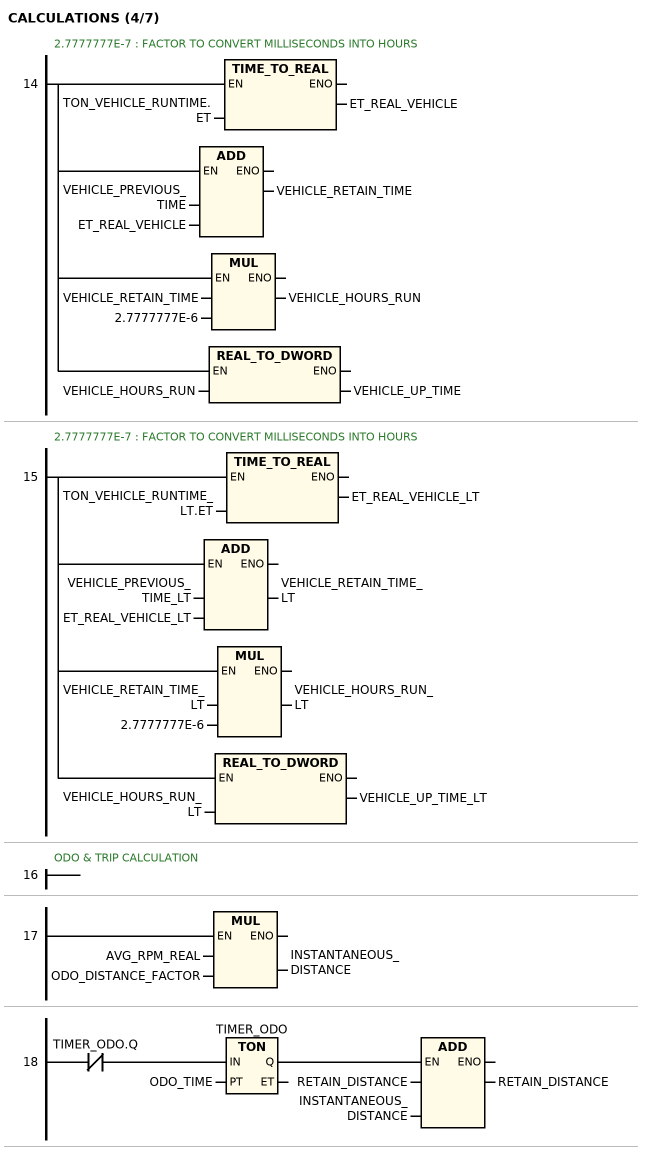
[picture p24: CALCULATIONS (LD)]
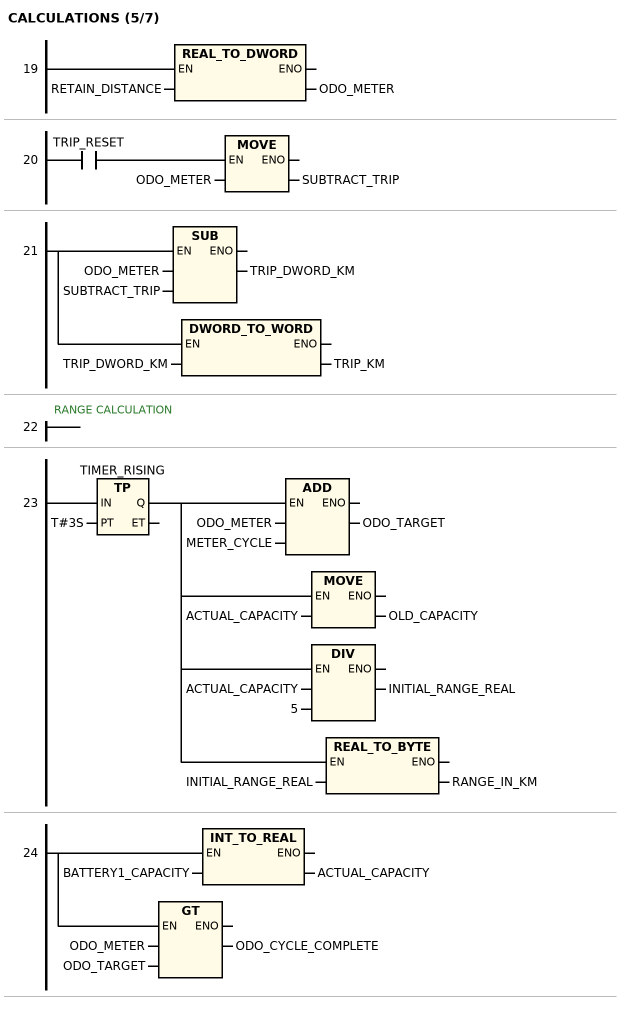
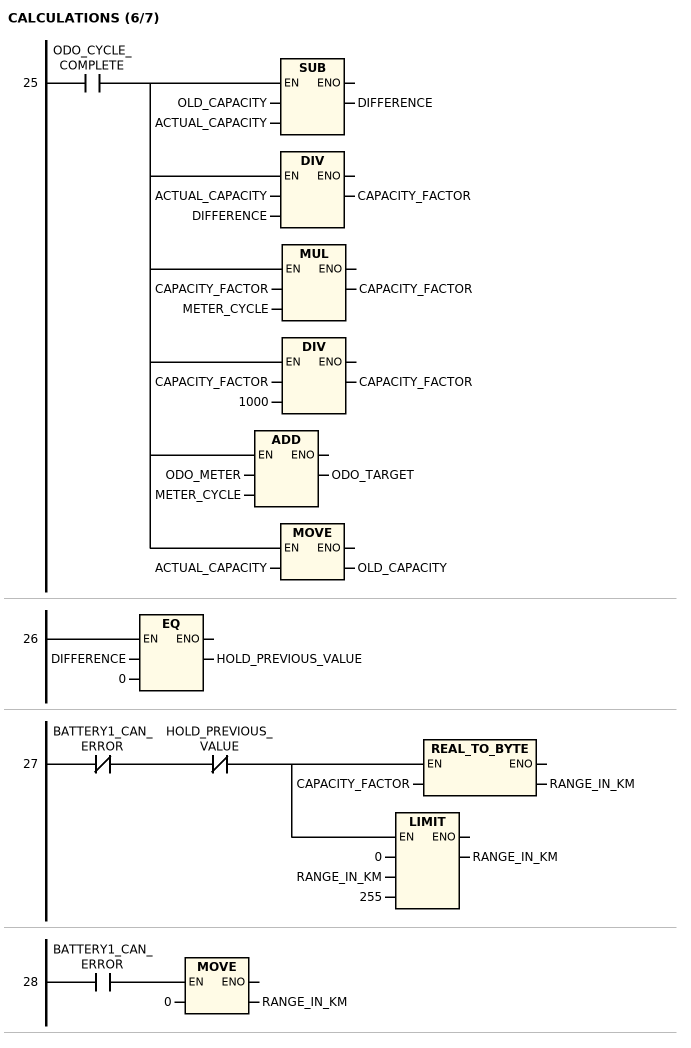
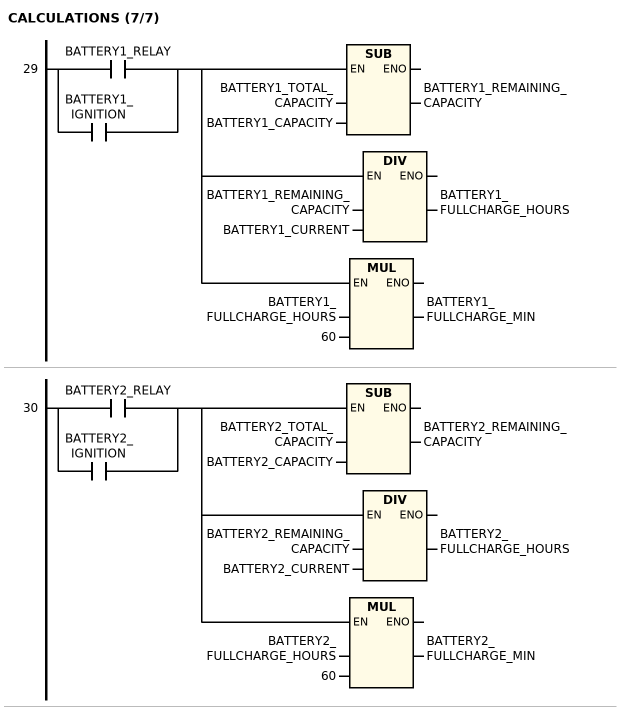
_LD_ (* Ladder Diagram *)
NETWORK 1 (* SPEED / GLX GEAR RATION = 72.02 / WHEEL DIA = 560 MM *)
	*
		EN --- ABS(MOTOR_RPM[1]) => ABS_RPM1
		EN --- ABS(MOTOR_RPM[2]) => ABS_RPM2
		EN --- ABS(MOTOR_RPM[6]) => ABS_RPM6
NETWORK 2
	*
		EN --- ADD(ABS_RPM1, ABS_RPM2) => RPM_SUM
		EN --- DIV(RPM_SUM, 2) => AVG_RPM
		EN --- ABS(AVG_RPM) => AVG_RPM
		EN --- INT_TO_REAL(AVG_RPM) => AVG_RPM_REAL
		EN --- MUL(AVG_RPM_REAL, SPEED_FACTOR) => SPEED_REAL
		EN --- REAL_TO_BYTE(SPEED_REAL) => SPEED
NETWORK 3 (* DRIVE AND HYDL UP TIME *)
	*
		EN --- GT(ABS_RPM1, 100) => MOTOR_1_RUNNING
		EN --- GT(ABS_RPM2, 100) => MOTOR_2_RUNNING
		EN --- OR(MOTOR_1_RUNNING, MOTOR_2_RUNNING) => COUNT_HOURS
		EN --- GT(ABS_RPM6, 100) => HYDRAULIC_HOURS
		EN --- OR(MCU_IGNITION, HYDRAULIC_SWITCH) => VEHICLE_UP_TIME_COUNT, VEHICLE_UP_TIME_COUNT_LT
NETWORK 4
	{ RISE:R_TRIG(CLK: *) | [COUNT_HOURS] - FALL:F_TRIG(CLK: *) }
		EN --- MOVE(RETAIN_TIME) => PREVIOUS_TIME
NETWORK 5
	{ RISE_2:R_TRIG(CLK: *) | [HYDRAULIC_HOURS] - FALL_2:F_TRIG(CLK: *) }
		EN --- MOVE(HYDL_RETAIN_TIME) => HYDL_PREVIOUS_TIME
NETWORK 6
	{ RISE_3:R_TRIG(CLK: *) | [VEHICLE_UP_TIME_COUNT] - FALL_3:F_TRIG(CLK: *) }
		EN --- MOVE(VEHICLE_RETAIN_TIME) => VEHICLE_PREVIOUS_TIME
NETWORK 7
	{ RISE_4:R_TRIG(CLK: *) | [VEHICLE_UP_TIME_COUNT_LT] - FALL_4:F_TRIG(CLK: *) }
		EN --- MOVE(VEHICLE_RETAIN_TIME_LT) => VEHICLE_PREVIOUS_TIME_LT
NETWORK 8
	[COUNT_HOURS] - TON_RUNTIME:TON(IN: *, PT: t#10d)
NETWORK 9
	[HYDRAULIC_HOURS] - TON_HYDL_RUNTIME:TON(IN: *, PT: t#10d)
NETWORK 10
	[VEHICLE_UP_TIME_COUNT] - TON_VEHICLE_RUNTIME:TON(IN: *, PT: t#10d)
NETWORK 11
	[VEHICLE_UP_TIME_COUNT_LT] - TON_VEHICLE_RUNTIME_LT:TON(IN: *, PT: t#10d)
NETWORK 12 (* 2.7777777E-6 : FACTOR TO CONVERT MILLISECONDS INTO (HOUR . MIN) (FACTOR IS 0.1) *)
	*
		EN --- TIME_TO_REAL(TON_RUNTIME.ET) => ET_REAL
		EN --- ADD(PREVIOUS_TIME, ET_REAL) => RETAIN_TIME
		EN --- MUL(RETAIN_TIME, 2.7777777E-6) => MINUTE_RUN
		EN --- REAL_TO_DWORD(MINUTE_RUN) => RUNTIME
NETWORK 13 (* 2.7777777E-7 : FACTOR TO CONVERT MILLISECONDS INTO HOURS *)
	*
		EN --- TIME_TO_REAL(TON_HYDL_RUNTIME.ET) => ET_REAL_HYDL
		EN --- ADD(HYDL_PREVIOUS_TIME, ET_REAL_HYDL) => HYDL_RETAIN_TIME
		EN --- MUL(HYDL_RETAIN_TIME, 2.7777777E-6) => HYDL_HOURS_RUN
		EN --- REAL_TO_DWORD(HYDL_HOURS_RUN) => HYDL_UP_TIME
NETWORK 14 (* 2.7777777E-7 : FACTOR TO CONVERT MILLISECONDS INTO HOURS *)
	*
		EN --- TIME_TO_REAL(TON_VEHICLE_RUNTIME.ET) => ET_REAL_VEHICLE
		EN --- ADD(VEHICLE_PREVIOUS_TIME, ET_REAL_VEHICLE) => VEHICLE_RETAIN_TIME
		EN --- MUL(VEHICLE_RETAIN_TIME, 2.7777777E-6) => VEHICLE_HOURS_RUN
		EN --- REAL_TO_DWORD(VEHICLE_HOURS_RUN) => VEHICLE_UP_TIME
NETWORK 15 (* 2.7777777E-7 : FACTOR TO CONVERT MILLISECONDS INTO HOURS *)
	*
		EN --- TIME_TO_REAL(TON_VEHICLE_RUNTIME_LT.ET) => ET_REAL_VEHICLE_LT
		EN --- ADD(VEHICLE_PREVIOUS_TIME_LT, ET_REAL_VEHICLE_LT) => VEHICLE_RETAIN_TIME_LT
		EN --- MUL(VEHICLE_RETAIN_TIME_LT, 2.7777777E-6) => VEHICLE_HOURS_RUN_LT
		EN --- REAL_TO_DWORD(VEHICLE_HOURS_RUN_LT) => VEHICLE_UP_TIME_LT
NETWORK 16 (* ODO & TRIP CALCULATION *)
	*
NETWORK 17
	*
		EN --- MUL(AVG_RPM_REAL, ODO_DISTANCE_FACTOR) => INSTANTANEOUS_DISTANCE
NETWORK 18
	[/TIMER_ODO.Q] - TIMER_ODO:TON(IN: *, PT: ODO_TIME)
		EN --- ADD(RETAIN_DISTANCE, INSTANTANEOUS_DISTANCE) => RETAIN_DISTANCE
NETWORK 19
	*
		EN --- REAL_TO_DWORD(RETAIN_DISTANCE) => ODO_METER
NETWORK 20
	[TRIP_RESET]
		EN --- MOVE(ODO_METER) => SUBTRACT_TRIP
NETWORK 21
	*
		EN --- SUB(ODO_METER, SUBTRACT_TRIP) => TRIP_DWORD_KM
		EN --- DWORD_TO_WORD(TRIP_DWORD_KM) => TRIP_KM
NETWORK 22 (* RANGE CALCULATION *)
	*
NETWORK 23
	TIMER_RISING:TP(IN: *, PT: T#3S)
		EN --- ADD(ODO_METER, METER_CYCLE) => ODO_TARGET
		EN --- MOVE(ACTUAL_CAPACITY) => OLD_CAPACITY
		EN --- DIV(ACTUAL_CAPACITY, 5) => INITIAL_RANGE_REAL
		EN --- REAL_TO_BYTE(INITIAL_RANGE_REAL) => RANGE_IN_KM
NETWORK 24
	*
		EN --- INT_TO_REAL(BATTERY1_CAPACITY) => ACTUAL_CAPACITY
		EN --- GT(ODO_METER, ODO_TARGET) => ODO_CYCLE_COMPLETE
NETWORK 25
	[ODO_CYCLE_COMPLETE]
		EN --- SUB(OLD_CAPACITY, ACTUAL_CAPACITY) => DIFFERENCE
		EN --- DIV(ACTUAL_CAPACITY, DIFFERENCE) => CAPACITY_FACTOR
		EN --- MUL(CAPACITY_FACTOR, METER_CYCLE) => CAPACITY_FACTOR
		EN --- DIV(CAPACITY_FACTOR, 1000) => CAPACITY_FACTOR
		EN --- ADD(ODO_METER, METER_CYCLE) => ODO_TARGET
		EN --- MOVE(ACTUAL_CAPACITY) => OLD_CAPACITY
NETWORK 26
	*
		EN --- EQ(DIFFERENCE, 0) => HOLD_PREVIOUS_VALUE
NETWORK 27
	[/BATTERY1_CAN_ERROR] - [/HOLD_PREVIOUS_VALUE]
		EN --- REAL_TO_BYTE(CAPACITY_FACTOR) => RANGE_IN_KM
		EN --- LIMIT(0, RANGE_IN_KM, 255) => RANGE_IN_KM
NETWORK 28
	[BATTERY1_CAN_ERROR]
		EN --- MOVE(0) => RANGE_IN_KM
NETWORK 29
	{ [BATTERY1_RELAY] | [BATTERY1_IGNITION] }
		EN --- SUB(BATTERY1_TOTAL_CAPACITY, BATTERY1_CAPACITY) => BATTERY1_REMAINING_CAPACITY
		EN --- DIV(BATTERY1_REMAINING_CAPACITY, BATTERY1_CURRENT) => BATTERY1_FULLCHARGE_HOURS
		EN --- MUL(BATTERY1_FULLCHARGE_HOURS, 60) => BATTERY1_FULLCHARGE_MIN
NETWORK 30
	{ [BATTERY2_RELAY] | [BATTERY2_IGNITION] }
		EN --- SUB(BATTERY2_TOTAL_CAPACITY, BATTERY2_CAPACITY) => BATTERY2_REMAINING_CAPACITY
		EN --- DIV(BATTERY2_REMAINING_CAPACITY, BATTERY2_CURRENT) => BATTERY2_FULLCHARGE_HOURS
		EN --- MUL(BATTERY2_FULLCHARGE_HOURS, 60) => BATTERY2_FULLCHARGE_MIN
_END_LD_
(* the same logic as Structured Text *)
(* Network 1 *)
ABS_RPM1 := ABS(MOTOR_RPM[1]);
ABS_RPM2 := ABS(MOTOR_RPM[2]);
ABS_RPM6 := ABS(MOTOR_RPM[6]);
(* Network 2 *)
RPM_SUM := ABS_RPM1 + ABS_RPM2;
AVG_RPM := RPM_SUM / 2;
AVG_RPM := ABS(AVG_RPM);
AVG_RPM_REAL := INT_TO_REAL(AVG_RPM);
SPEED_REAL := AVG_RPM_REAL * SPEED_FACTOR;
SPEED := REAL_TO_BYTE(SPEED_REAL);
(* Network 3: see the listing above *)
(* Network 4 *)
RISE(CLK := TRUE);
FALL(CLK := COUNT_HOURS);
IF RISE.Q OR FALL.Q THEN
	PREVIOUS_TIME := RETAIN_TIME;
END_IF;
(* Network 5 *)
RISE_2(CLK := TRUE);
FALL_2(CLK := HYDRAULIC_HOURS);
IF RISE_2.Q OR FALL_2.Q THEN
	HYDL_PREVIOUS_TIME := HYDL_RETAIN_TIME;
END_IF;
(* Network 6 *)
RISE_3(CLK := TRUE);
FALL_3(CLK := VEHICLE_UP_TIME_COUNT);
IF RISE_3.Q OR FALL_3.Q THEN
	VEHICLE_PREVIOUS_TIME := VEHICLE_RETAIN_TIME;
END_IF;
(* Network 7 *)
RISE_4(CLK := TRUE);
FALL_4(CLK := VEHICLE_UP_TIME_COUNT_LT);
IF RISE_4.Q OR FALL_4.Q THEN
	VEHICLE_PREVIOUS_TIME_LT := VEHICLE_RETAIN_TIME_LT;
END_IF;
(* Network 8 *)
TON_RUNTIME(IN := COUNT_HOURS, PT := t#10d);
(* Network 9 *)
TON_HYDL_RUNTIME(IN := HYDRAULIC_HOURS, PT := t#10d);
(* Network 10 *)
TON_VEHICLE_RUNTIME(IN := VEHICLE_UP_TIME_COUNT, PT := t#10d);
(* Network 11 *)
TON_VEHICLE_RUNTIME_LT(IN := VEHICLE_UP_TIME_COUNT_LT, PT := t#10d);
(* Network 12 *)
ET_REAL := TIME_TO_REAL(TON_RUNTIME.ET);
RETAIN_TIME := PREVIOUS_TIME + ET_REAL;
MINUTE_RUN := RETAIN_TIME * (2.7777777E-6);
RUNTIME := REAL_TO_DWORD(MINUTE_RUN);
(* Network 13 *)
ET_REAL_HYDL := TIME_TO_REAL(TON_HYDL_RUNTIME.ET);
HYDL_RETAIN_TIME := HYDL_PREVIOUS_TIME + ET_REAL_HYDL;
HYDL_HOURS_RUN := HYDL_RETAIN_TIME * (2.7777777E-6);
HYDL_UP_TIME := REAL_TO_DWORD(HYDL_HOURS_RUN);
(* Network 14 *)
ET_REAL_VEHICLE := TIME_TO_REAL(TON_VEHICLE_RUNTIME.ET);
VEHICLE_RETAIN_TIME := VEHICLE_PREVIOUS_TIME + ET_REAL_VEHICLE;
VEHICLE_HOURS_RUN := VEHICLE_RETAIN_TIME * (2.7777777E-6);
VEHICLE_UP_TIME := REAL_TO_DWORD(VEHICLE_HOURS_RUN);
(* Network 15 *)
ET_REAL_VEHICLE_LT := TIME_TO_REAL(TON_VEHICLE_RUNTIME_LT.ET);
VEHICLE_RETAIN_TIME_LT := VEHICLE_PREVIOUS_TIME_LT + ET_REAL_VEHICLE_LT;
VEHICLE_HOURS_RUN_LT := VEHICLE_RETAIN_TIME_LT * (2.7777777E-6);
VEHICLE_UP_TIME_LT := REAL_TO_DWORD(VEHICLE_HOURS_RUN_LT);
(* Network 16: see the listing above *)
(* Network 17 *)
INSTANTANEOUS_DISTANCE := AVG_RPM_REAL * ODO_DISTANCE_FACTOR;
(* Network 18 *)
TIMER_ODO(IN := NOT TIMER_ODO.Q, PT := ODO_TIME);
IF TIMER_ODO.Q THEN
	RETAIN_DISTANCE := RETAIN_DISTANCE + INSTANTANEOUS_DISTANCE;
END_IF;
(* Network 19 *)
ODO_METER := REAL_TO_DWORD(RETAIN_DISTANCE);
(* Network 20 *)
IF TRIP_RESET THEN
	SUBTRACT_TRIP := ODO_METER;
END_IF;
(* Network 21 *)
TRIP_DWORD_KM := ODO_METER - SUBTRACT_TRIP;
TRIP_KM := DWORD_TO_WORD(TRIP_DWORD_KM);
(* Network 22: see the listing above *)
(* Network 23 *)
TIMER_RISING(IN := TRUE, PT := T#3S);
IF TIMER_RISING.Q THEN
	ODO_TARGET := ODO_METER + METER_CYCLE;
	OLD_CAPACITY := ACTUAL_CAPACITY;
	INITIAL_RANGE_REAL := ACTUAL_CAPACITY / 5;
	RANGE_IN_KM := REAL_TO_BYTE(INITIAL_RANGE_REAL);
END_IF;
(* Network 24 *)
ACTUAL_CAPACITY := INT_TO_REAL(BATTERY1_CAPACITY);
ODO_CYCLE_COMPLETE := ODO_METER > ODO_TARGET;
(* Network 25 *)
IF ODO_CYCLE_COMPLETE THEN
	DIFFERENCE := OLD_CAPACITY - ACTUAL_CAPACITY;
	CAPACITY_FACTOR := ACTUAL_CAPACITY / DIFFERENCE;
	CAPACITY_FACTOR := CAPACITY_FACTOR * METER_CYCLE;
	CAPACITY_FACTOR := CAPACITY_FACTOR / 1000;
	ODO_TARGET := ODO_METER + METER_CYCLE;
	OLD_CAPACITY := ACTUAL_CAPACITY;
END_IF;
(* Network 26 *)
HOLD_PREVIOUS_VALUE := DIFFERENCE = 0;
(* Network 27 *)
IF NOT BATTERY1_CAN_ERROR AND NOT HOLD_PREVIOUS_VALUE THEN
	RANGE_IN_KM := REAL_TO_BYTE(CAPACITY_FACTOR);
	RANGE_IN_KM := LIMIT(0, RANGE_IN_KM, 255);
END_IF;
(* Network 28 *)
IF BATTERY1_CAN_ERROR THEN
	RANGE_IN_KM := 0;
END_IF;
(* Network 29 *)
IF BATTERY1_RELAY OR BATTERY1_IGNITION THEN
	BATTERY1_REMAINING_CAPACITY := BATTERY1_TOTAL_CAPACITY - BATTERY1_CAPACITY;
	BATTERY1_FULLCHARGE_HOURS := BATTERY1_REMAINING_CAPACITY / BATTERY1_CURRENT;
	BATTERY1_FULLCHARGE_MIN := BATTERY1_FULLCHARGE_HOURS * 60;
END_IF;
(* Network 30 *)
IF BATTERY2_RELAY OR BATTERY2_IGNITION THEN
	BATTERY2_REMAINING_CAPACITY := BATTERY2_TOTAL_CAPACITY - BATTERY2_CAPACITY;
	BATTERY2_FULLCHARGE_HOURS := BATTERY2_REMAINING_CAPACITY / BATTERY2_CURRENT;
	BATTERY2_FULLCHARGE_MIN := BATTERY2_FULLCHARGE_HOURS * 60;
END_IF;
END_PROGRAM

(* POU FB_LIBRARY/ALTERNATE, LD *)
FUNCTION_BLOCK ALTERNATE
VAR_INPUT
	IN: BOOL;
END_VAR
VAR_OUTPUT
	OUT: BOOL;
END_VAR
VAR
	S1: BOOL;
	S2: BOOL;
END_VAR
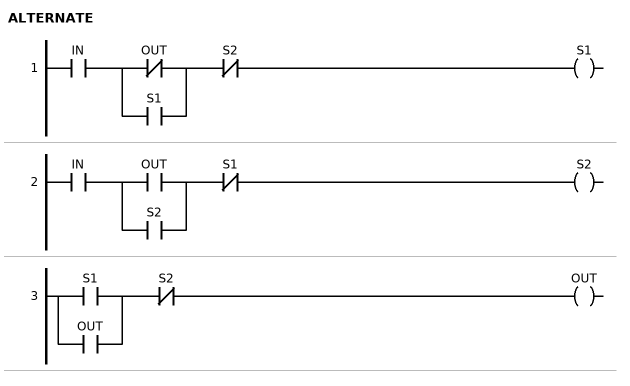
_LD_ (* Ladder Diagram *)
NETWORK 1
	[IN] - { [/OUT] | [S1] } - [/S2] --- (S1)
NETWORK 2
	[IN] - { [OUT] | [S2] } - [/S1] --- (S2)
NETWORK 3
	{ [S1] | [OUT] } - [/S2] --- (OUT)
_END_LD_
(* the same logic as Structured Text *)
(* Network 1 *)
S1 := IN AND (NOT OUT OR S1) AND NOT S2;
(* Network 2 *)
S2 := IN AND (OUT OR S2) AND NOT S1;
(* Network 3 *)
OUT := (S1 OR OUT) AND NOT S2;
END_FUNCTION_BLOCK

(* POU PROGRAM_FBs/ARM_LOGIC, LD *)
FUNCTION_BLOCK ARM_LOGIC
VAR_INPUT
	ARM_INPUT: BOOL;
	DISARM: BOOL;
	POST_IN: BOOL;
END_VAR
VAR_OUTPUT
	ARM: BOOL;
	ARMLED: BOOL;
END_VAR
VAR
	DELAY: TON;
	S1: BOOL;
	S2: BOOL;
	BLINKY: BLINK;
END_VAR
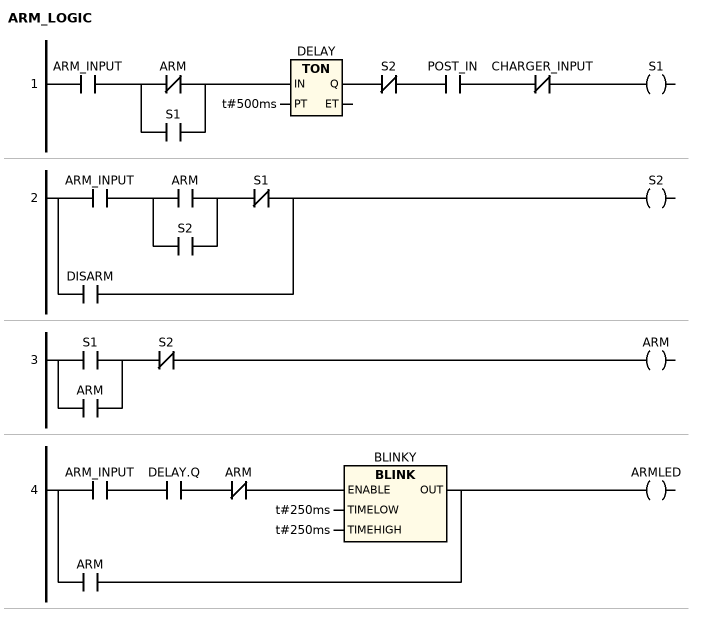
_LD_ (* Ladder Diagram *)
NETWORK 1
	[ARM_INPUT] - { [/ARM] | [S1] } - DELAY:TON(IN: *, PT: t#500ms) - [/S2] - [POST_IN] - [/CHARGER_INPUT] --- (S1)
NETWORK 2
	{ [ARM_INPUT] - { [ARM] | [S2] } - [/S1] | [DISARM] } --- (S2)
NETWORK 3
	{ [S1] | [ARM] } - [/S2] --- (ARM)
NETWORK 4
	{ [ARM_INPUT] - [DELAY.Q] - [/ARM] - BLINKY:BLINK(ENABLE: *, TIMELOW: t#250ms, TIMEHIGH: t#250ms) | [ARM] } --- (ARMLED)
_END_LD_
(* the same logic as Structured Text *)
(* Network 1 *)
DELAY(IN := ARM_INPUT AND (NOT ARM OR S1), PT := t#500ms);
S1 := DELAY.Q AND NOT S2 AND POST_IN AND NOT CHARGER_INPUT;
(* Network 2 *)
S2 := ARM_INPUT AND (ARM OR S2) AND NOT S1 OR DISARM;
(* Network 3 *)
ARM := (S1 OR ARM) AND NOT S2;
(* Network 4 *)
BLINKY(ENABLE := ARM_INPUT AND DELAY.Q AND NOT ARM, TIMELOW := t#250ms, TIMEHIGH := t#250ms);
ARMLED := BLINKY.OUT OR ARM;
END_FUNCTION_BLOCK

(* POU FUNCTIONS/BYTE_WORD_FUNCTION, ST *)
FUNCTION BYTE_WORD_FUNCTION : WORD
(*
Created by: Bhagyesh Unadkat
Date: 29-03-24
Version: 1
Updated by:
Update date:
Description: This block merges Two bytes of data into WORD data.
*)
VAR_INPUT
	BYTE_H: BYTE;
	BYTE_L: BYTE;
END_VAR
VAR
	MSB: WORD;
END_VAR
MSB:= BYTE_H * 256;
BYTE_WORD_FUNCTION:= MSB + BYTE_L;
END_FUNCTION

(* POU MCU/CHARA_MCU_RX, LD *)
FUNCTION_BLOCK CHARA_MCU_RX
(*
Created by: Bhagyesh Unadkat
Date: 11-09-24
Version: 5
Updated by: Karthik
Update date: 08-03-25
Description: This block receives CAN data from CHARA MCU.

		***Updates***
V2
	DC current and POWER added.
V3   
	Added OBD Code and adjusted the fault array accordingly.
	CAN error added to OBD code MSB bit as it is 12-bit value.
V4 
	Taken Motor Ignition as VAR_INPUT to reset RPM AND POWER TO 0
V5
	Converted CURRENT raw values from word to int, and then dividing by 1000.
V6
	Unmerged CAN error and OBD code.
V7
	Making OBD code zero when theres is a CAN error. 

FAULT ARRAY [DATATYPE: BYTE]
[1] MSG-2 BYTE2 and MSG-5 BYTE3		
		BYTE [BIT 0..7]: MSG2BYTE2 (BIT_0 TO BIT_2)------- AND-------- MSG5BYTE3 (BIT_0 TO BIT_4)
[2] MSG 2 :BYTE 7
[3] MSG 5: BYTE 2
[4] MSG 5: BYTE 4
*)
VAR_INPUT
	IGNITION: BOOL;
	MOTOR_IGNITION: BOOL;
	CAN_CHANNEL: BYTE;
	ID_1: DWORD;
	ID_2: DWORD;
	ID_4: DWORD;
	ID_5: DWORD;
	ID_6: DWORD;
END_VAR
VAR_OUTPUT
	RPM: INT;
	POWER: INT;
	PHASE_CURRENT: WORD;
	M_TEMP: BYTE;
	C_TEMP: BYTE;
	OBD_CODE: WORD;
	FAULT_ARRAY: ARRAY [1..4] OF BYTE;
	CAN_ERROR: BOOL;
END_VAR
VAR
	RX_1: RX_CAN;
	RX_2: RX_CAN;
	RX_4: RX_CAN;
	RX_5: RX_CAN;
	RX_6: RX_CAN;
	TIMER_ERROR: TON;

	RPM_WORD: WORD;
	PHASE_WORD: WORD;
	REVERSE_DIRECTION: BOOL;
	DIR_FACTOR: INT;
	DELAY: TON;
	RPM_INT: INT;
	CURRENT_WORD: WORD;
	CURRENT_INT: INT;
	VOLTAGE_INT: INT;
	RPM_SIGNED: INT;
	POWER_INT: INT;
END_VAR
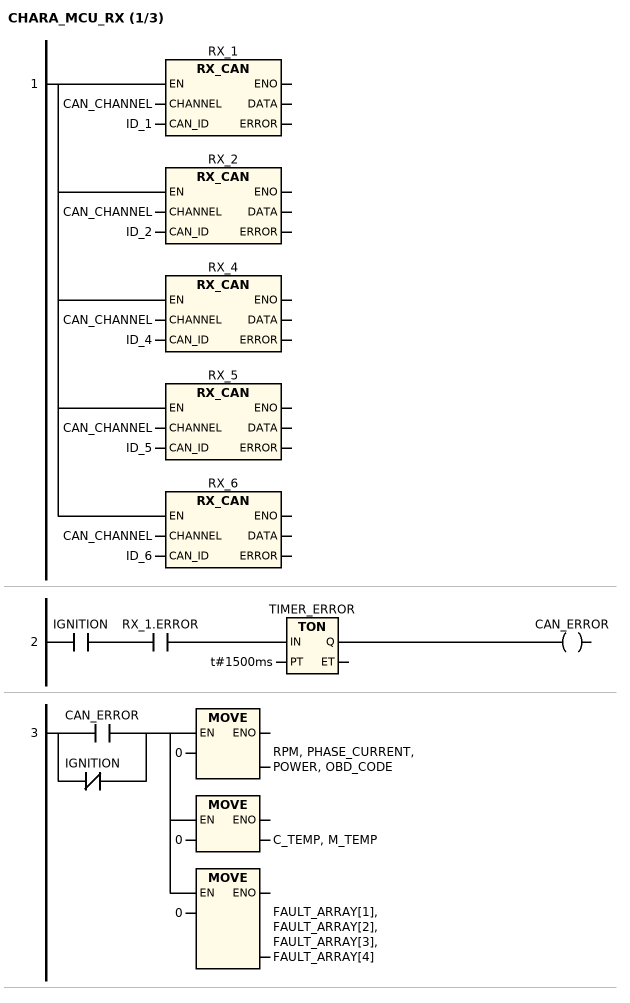
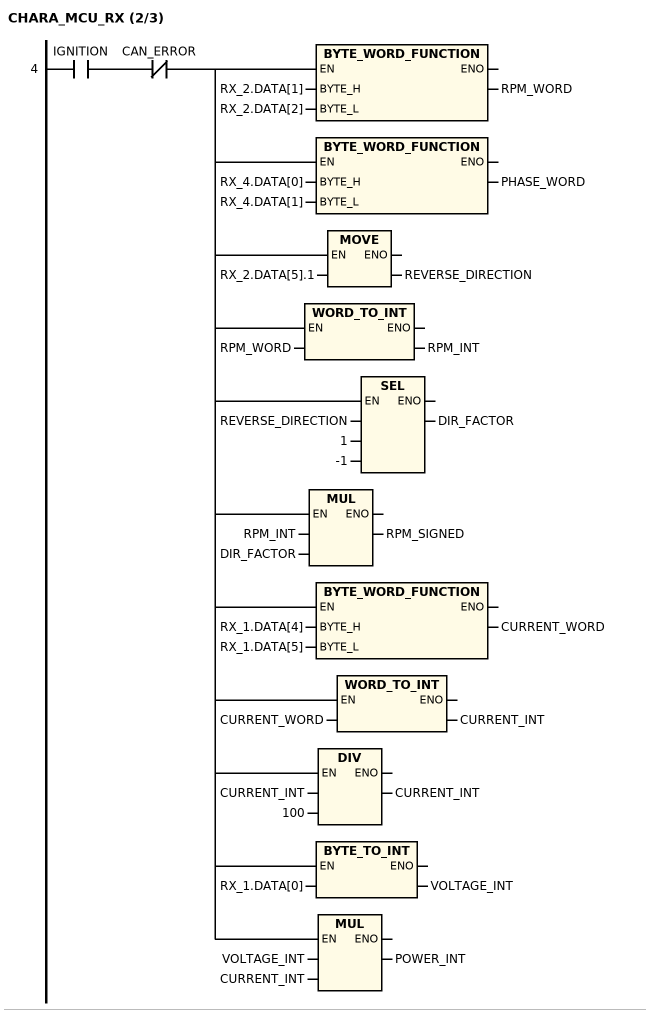
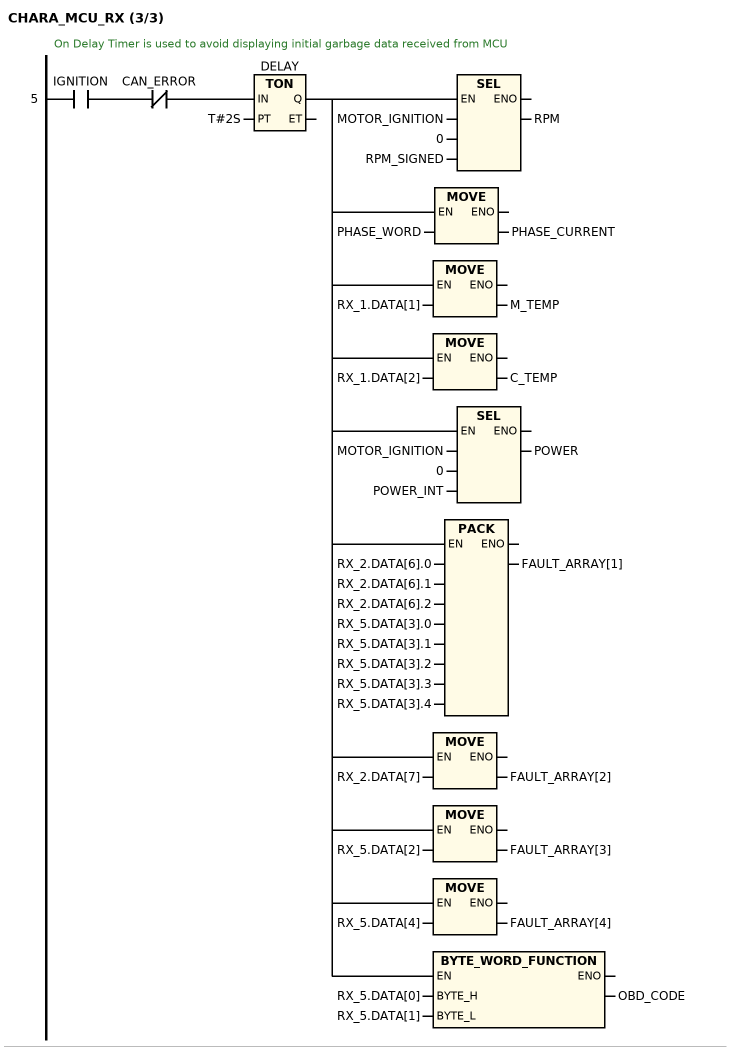
_LD_ (* Ladder Diagram *)
NETWORK 1
	*
		EN --- RX_1:RX_CAN(CHANNEL: CAN_CHANNEL, CAN_ID: ID_1)
		EN --- RX_2:RX_CAN(CHANNEL: CAN_CHANNEL, CAN_ID: ID_2)
		EN --- RX_4:RX_CAN(CHANNEL: CAN_CHANNEL, CAN_ID: ID_4)
		EN --- RX_5:RX_CAN(CHANNEL: CAN_CHANNEL, CAN_ID: ID_5)
		EN --- RX_6:RX_CAN(CHANNEL: CAN_CHANNEL, CAN_ID: ID_6)
NETWORK 2
	[IGNITION] - [RX_1.ERROR] - TIMER_ERROR:TON(IN: *, PT: t#1500ms) --- (CAN_ERROR)
NETWORK 3
	{ [CAN_ERROR] | [/IGNITION] }
		EN --- MOVE(0) => RPM, PHASE_CURRENT, POWER, OBD_CODE
		EN --- MOVE(0) => C_TEMP, M_TEMP
		EN --- MOVE(0) => FAULT_ARRAY[1], FAULT_ARRAY[2], FAULT_ARRAY[3], FAULT_ARRAY[4]
NETWORK 4
	[IGNITION] - [/CAN_ERROR]
		EN --- BYTE_WORD_FUNCTION(BYTE_H: RX_2.DATA[1], BYTE_L: RX_2.DATA[2]) => RPM_WORD
		EN --- BYTE_WORD_FUNCTION(BYTE_H: RX_4.DATA[0], BYTE_L: RX_4.DATA[1]) => PHASE_WORD
		EN --- MOVE(RX_2.DATA[5].1) => REVERSE_DIRECTION
		EN --- WORD_TO_INT(RPM_WORD) => RPM_INT
		EN --- SEL(REVERSE_DIRECTION, 1, -1) => DIR_FACTOR
		EN --- MUL(RPM_INT, DIR_FACTOR) => RPM_SIGNED
		EN --- BYTE_WORD_FUNCTION(BYTE_H: RX_1.DATA[4], BYTE_L: RX_1.DATA[5]) => CURRENT_WORD
		EN --- WORD_TO_INT(CURRENT_WORD) => CURRENT_INT
		EN --- DIV(CURRENT_INT, 100) => CURRENT_INT
		EN --- BYTE_TO_INT(RX_1.DATA[0]) => VOLTAGE_INT
		EN --- MUL(VOLTAGE_INT, CURRENT_INT) => POWER_INT
NETWORK 5 (* On Delay Timer is used to avoid displaying initial garbage data received from MCU *)
	[IGNITION] - [/CAN_ERROR] - DELAY:TON(IN: *, PT: T#2S)
		EN --- SEL(MOTOR_IGNITION, 0, RPM_SIGNED) => RPM
		EN --- MOVE(PHASE_WORD) => PHASE_CURRENT
		EN --- MOVE(RX_1.DATA[1]) => M_TEMP
		EN --- MOVE(RX_1.DATA[2]) => C_TEMP
		EN --- SEL(MOTOR_IGNITION, 0, POWER_INT) => POWER
		EN --- PACK(RX_2.DATA[6].0, RX_2.DATA[6].1, RX_2.DATA[6].2, RX_5.DATA[3].0, RX_5.DATA[3].1, RX_5.DATA[3].2, RX_5.DATA[3].3, RX_5.DATA[3].4) => FAULT_ARRAY[1]
		EN --- MOVE(RX_2.DATA[7]) => FAULT_ARRAY[2]
		EN --- MOVE(RX_5.DATA[2]) => FAULT_ARRAY[3]
		EN --- MOVE(RX_5.DATA[4]) => FAULT_ARRAY[4]
		EN --- BYTE_WORD_FUNCTION(BYTE_H: RX_5.DATA[0], BYTE_L: RX_5.DATA[1]) => OBD_CODE
_END_LD_
(* the same logic as Structured Text *)
(* Network 1 *)
RX_1(CHANNEL := CAN_CHANNEL, CAN_ID := ID_1);
RX_2(CHANNEL := CAN_CHANNEL, CAN_ID := ID_2);
RX_4(CHANNEL := CAN_CHANNEL, CAN_ID := ID_4);
RX_5(CHANNEL := CAN_CHANNEL, CAN_ID := ID_5);
RX_6(CHANNEL := CAN_CHANNEL, CAN_ID := ID_6);
(* Network 2 *)
TIMER_ERROR(IN := IGNITION AND RX_1.ERROR, PT := t#1500ms);
CAN_ERROR := TIMER_ERROR.Q;
(* Network 3: see the listing above *)
(* Network 4 *)
IF IGNITION AND NOT CAN_ERROR THEN
	RPM_WORD := BYTE_WORD_FUNCTION(BYTE_H := RX_2.DATA[1], BYTE_L := RX_2.DATA[2]);
	PHASE_WORD := BYTE_WORD_FUNCTION(BYTE_H := RX_4.DATA[0], BYTE_L := RX_4.DATA[1]);
	REVERSE_DIRECTION := RX_2.DATA[5].1;
	RPM_INT := WORD_TO_INT(RPM_WORD);
	DIR_FACTOR := SEL(REVERSE_DIRECTION, 1, -1);
	RPM_SIGNED := RPM_INT * DIR_FACTOR;
	CURRENT_WORD := BYTE_WORD_FUNCTION(BYTE_H := RX_1.DATA[4], BYTE_L := RX_1.DATA[5]);
	CURRENT_INT := WORD_TO_INT(CURRENT_WORD);
	CURRENT_INT := CURRENT_INT / 100;
	VOLTAGE_INT := BYTE_TO_INT(RX_1.DATA[0]);
	POWER_INT := VOLTAGE_INT * CURRENT_INT;
END_IF;
(* Network 5 *)
DELAY(IN := IGNITION AND NOT CAN_ERROR, PT := T#2S);
IF DELAY.Q THEN
	RPM := SEL(MOTOR_IGNITION, 0, RPM_SIGNED);
	PHASE_CURRENT := PHASE_WORD;
	M_TEMP := RX_1.DATA[1];
	C_TEMP := RX_1.DATA[2];
	POWER := SEL(MOTOR_IGNITION, 0, POWER_INT);
	FAULT_ARRAY[1] := PACK(RX_2.DATA[6].0, RX_2.DATA[6].1, RX_2.DATA[6].2, RX_5.DATA[3].0, RX_5.DATA[3].1, RX_5.DATA[3].2, RX_5.DATA[3].3, RX_5.DATA[3].4);
	FAULT_ARRAY[2] := RX_2.DATA[7];
	FAULT_ARRAY[3] := RX_5.DATA[2];
	FAULT_ARRAY[4] := RX_5.DATA[4];
	OBD_CODE := BYTE_WORD_FUNCTION(BYTE_H := RX_5.DATA[0], BYTE_L := RX_5.DATA[1]);
END_IF;
END_FUNCTION_BLOCK

(* POU MCU/CHARA_MCU_TX, LD *)
FUNCTION_BLOCK CHARA_MCU_TX
(*
Created by: Bhagyesh Unadkat
Date: Sep 11, 2024
Version: 4
Updated by: Bhagyesh
Update date: Dec 13, 2024
Description: This block transmits CAN data to the CHARA MCU to control the motor.

NOTE:  BIG ENDIAN FORMAT

Byte0 & Byte1: Signed RPM Big Endian format (-6000 to 6000)
Byte2: Ignition State =  0 & 1 (OFF and ON respectively)
Byte3: Phase Current Limit (%) = 0 - 100
Byte4: Regen (%) = 0 - 100 (Not configured yet)
Byte5: Acceleration time (s) = 1 unit is 100ms
Byte6: Deceleration time (s) =  1 unit is 100ms

CAN ID X value for the different Node ID:
41 - 9		42 - A 		43-B
	
	***UPDATES***
V2:
1. RPM transmit delay has been added after Ignition turns on..
2. CAN_TX block has been changerd to CAN_TX_ENH.
3. Temporary Phase current limit has been added to var input
V3
1. Added Ignition state bit as VAR_OUTPUT.
V4
1. UPDATED AVG RPM TO 75 TO HOLD ON THE MCU.
2. RPM DELAY TIME REDUCED TO 250MS
*)
VAR_INPUT
	CAN_CHANNEL: BYTE;
	ID_22X: DWORD;
	TARGET_RPM: INT;
	REFERNCE_RPM: INT;
	RAMP: INT;
	MCU_RAMP: BYTE;
	HILL_HOLD_IN: BOOL;
	PHASE_CURRENT_LIMIT: BYTE;
END_VAR
VAR
	IGNITION_ON: BOOL;
	IGNITION_STATE: BYTE;
	HOLD_ON: BOOL;
	ABS_RPM: INT;
	RPM_RAMP: RAMP_INT;
	WB_TARGET_RPM: WORD_BYTE_CONVERSION;
	PACK_TX: PACK_BYTES;
	TX: CAN_TX_ENH;
	RPM_DELAY: TON;
	TIMER: TON;
END_VAR
VAR_OUTPUT
	TARGET_RPM_OUT: INT;
	IGNITION_OUT: BOOL;
END_VAR
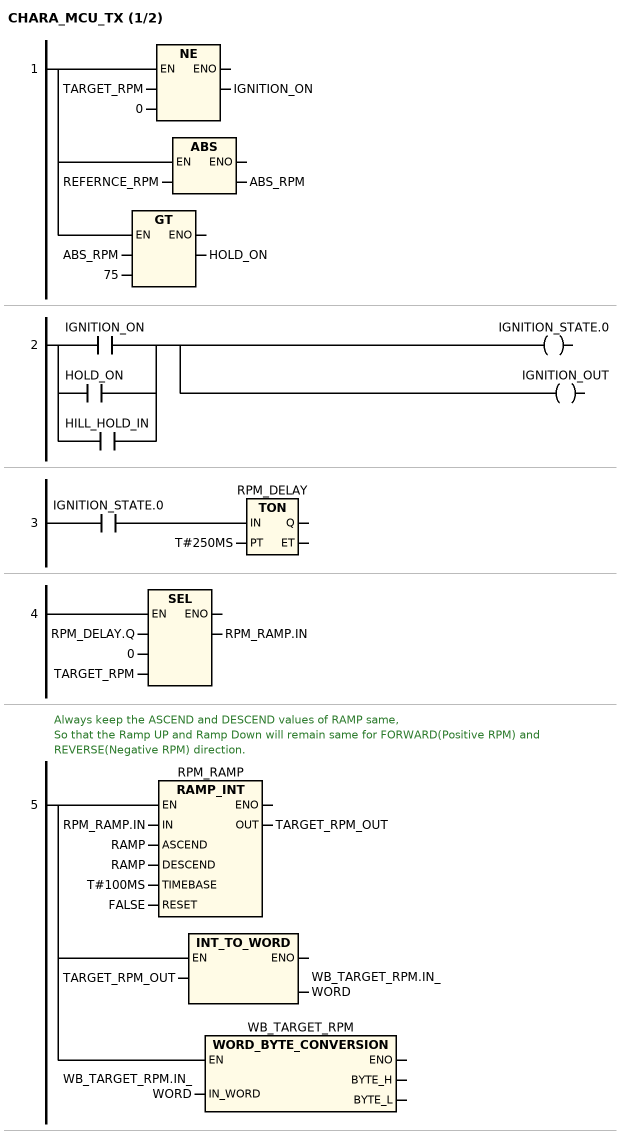
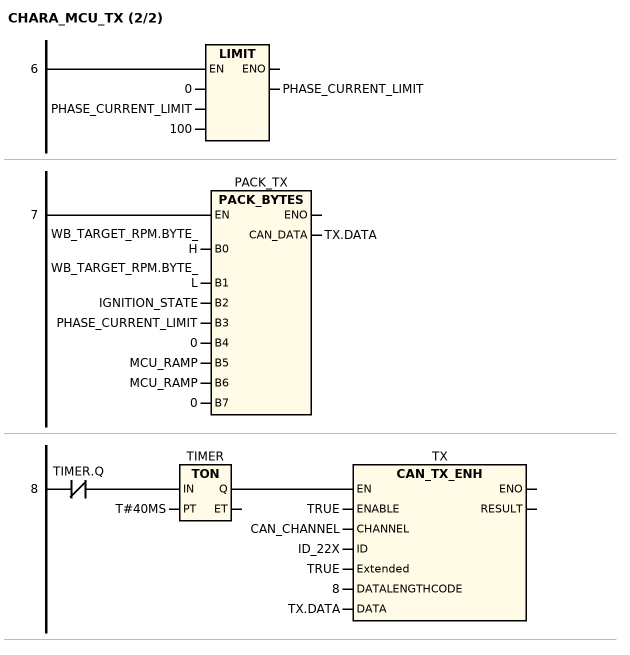
_LD_ (* Ladder Diagram *)
NETWORK 1
	*
		EN --- NE(TARGET_RPM, 0) => IGNITION_ON
		EN --- ABS(REFERNCE_RPM) => ABS_RPM
		EN --- GT(ABS_RPM, 75) => HOLD_ON
NETWORK 2
	{ [IGNITION_ON] | [HOLD_ON] | [HILL_HOLD_IN] } --- (IGNITION_STATE.0) (IGNITION_OUT)
NETWORK 3
	[IGNITION_STATE.0] - RPM_DELAY:TON(IN: *, PT: T#250MS)
NETWORK 4
	*
		EN --- SEL(RPM_DELAY.Q, 0, TARGET_RPM) => RPM_RAMP.IN
NETWORK 5 (* Always keep the ASCEND and DESCEND values of RAMP same, / So that the Ramp UP and Ramp Down will remain same for FORWARD(Positive RPM) and REVERSE(Negative RPM) direction. *)
	*
		EN --- RPM_RAMP:RAMP_INT(IN: RPM_RAMP.IN, ASCEND: RAMP, DESCEND: RAMP, TIMEBASE: T#100MS, RESET: FALSE) => TARGET_RPM_OUT
		EN --- INT_TO_WORD(TARGET_RPM_OUT) => WB_TARGET_RPM.IN_WORD
		EN --- WB_TARGET_RPM:WORD_BYTE_CONVERSION(IN_WORD: WB_TARGET_RPM.IN_WORD)
NETWORK 6
	*
		EN --- LIMIT(0, PHASE_CURRENT_LIMIT, 100) => PHASE_CURRENT_LIMIT
NETWORK 7
	*
		EN --- PACK_TX:PACK_BYTES(B0: WB_TARGET_RPM.BYTE_H, B1: WB_TARGET_RPM.BYTE_L, B2: IGNITION_STATE, B3: PHASE_CURRENT_LIMIT, B4: 0, B5: MCU_RAMP, B6: MCU_RAMP, B7: 0) => TX.DATA
NETWORK 8
	[/TIMER.Q] - TIMER:TON(IN: *, PT: T#40MS)
		EN --- TX:CAN_TX_ENH(ENABLE: TRUE, CHANNEL: CAN_CHANNEL, ID: ID_22X, Extended: TRUE, DATALENGTHCODE: 8, DATA: TX.DATA)
_END_LD_
(* the same logic as Structured Text *)
(* Network 1 *)
IGNITION_ON := TARGET_RPM <> 0;
ABS_RPM := ABS(REFERNCE_RPM);
HOLD_ON := ABS_RPM > 75;
(* Network 2 *)
IGNITION_STATE.0 := IGNITION_ON OR HOLD_ON OR HILL_HOLD_IN;
IGNITION_OUT := IGNITION_STATE.0;
(* Network 3 *)
RPM_DELAY(IN := IGNITION_STATE.0, PT := T#250MS);
(* Network 4 *)
RPM_RAMP.IN := SEL(RPM_DELAY.Q, 0, TARGET_RPM);
(* Network 5: Always keep the ASCEND and DESCEND values of RAMP same, / So that the Ramp UP and Ramp Down will remain same for FORWARD(Positive RPM) and REVERSE(Negative RPM) direction. *)
RPM_RAMP(IN := RPM_RAMP.IN, ASCEND := RAMP, DESCEND := RAMP, TIMEBASE := T#100MS, RESET := FALSE);
TARGET_RPM_OUT := RPM_RAMP.OUT;
WB_TARGET_RPM.IN_WORD := INT_TO_WORD(TARGET_RPM_OUT);
WB_TARGET_RPM(IN_WORD := WB_TARGET_RPM.IN_WORD);
(* Network 6 *)
PHASE_CURRENT_LIMIT := LIMIT(0, PHASE_CURRENT_LIMIT, 100);
(* Network 7 *)
PACK_TX(B0 := WB_TARGET_RPM.BYTE_H, B1 := WB_TARGET_RPM.BYTE_L, B2 := IGNITION_STATE, B3 := PHASE_CURRENT_LIMIT, B4 := 0, B5 := MCU_RAMP, B6 := MCU_RAMP, B7 := 0);
TX.DATA := PACK_TX.CAN_DATA;
(* Network 8 *)
TIMER(IN := NOT TIMER.Q, PT := T#40MS);
IF TIMER.Q THEN
	TX(ENABLE := TRUE, CHANNEL := CAN_CHANNEL, ID := ID_22X, Extended := TRUE, DATALENGTHCODE := 8, DATA := TX.DATA);
END_IF;
END_FUNCTION_BLOCK

(* POU PROGRAM_FBs/CLN_BATTERY, LD *)
FUNCTION_BLOCK CLN_BATTERY
(*
Created by: Anirudh Raghavan
Date: 10-01-24
Version: 4
Updated by: Bhagyesh
Update date: 15-09-2024
Description: This block reads the data of CLN Battery.
	
	*** UPDATES ***
V3: 
	Removed the SOC mapping function.
V4
	Variable modifiacations and faults removed
*)
VAR_INPUT
	CAN_CHANNEL: BYTE;
END_VAR
VAR_OUTPUT
	SOC: BYTE;
	SOH: BYTE;
       CURRENT: INT;
	CHARGING: BOOL;
	POWER: INT; (*Watt*)
	NTC_1: BYTE;
	NTC_2: BYTE;
	TOTAL_CAPACITY: INT; (*Ah*)
	CAPACITY: INT; (*Ah*)
	CAN_ERROR: BOOL;

END_VAR
VAR
	RX_205: RX_CAN;
	RX_1E1: RX_CAN;
	RX_1F5: RX_CAN;
	RX_357: RX_CAN;
	DELAY: TON;
	SOC_WORD: WORD;
	SOH_WORD: WORD;
	VOLTAGE_WORD: WORD;
	CURRENT_WORD: WORD;
	VOLTAGE: INT;
	CAPACITY_WORD: WORD;
	CAPACITY_AH: WORD;
	TOTAL_CAPACITY_WORD: WORD;
	TOTAL_CAPACITY_AH: WORD;

END_VAR
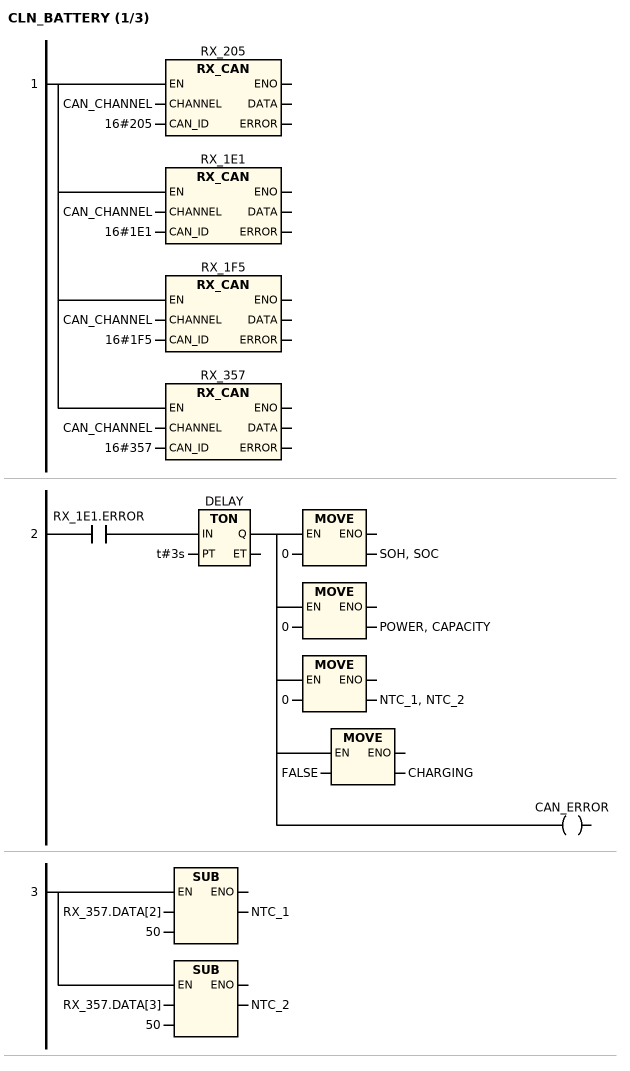
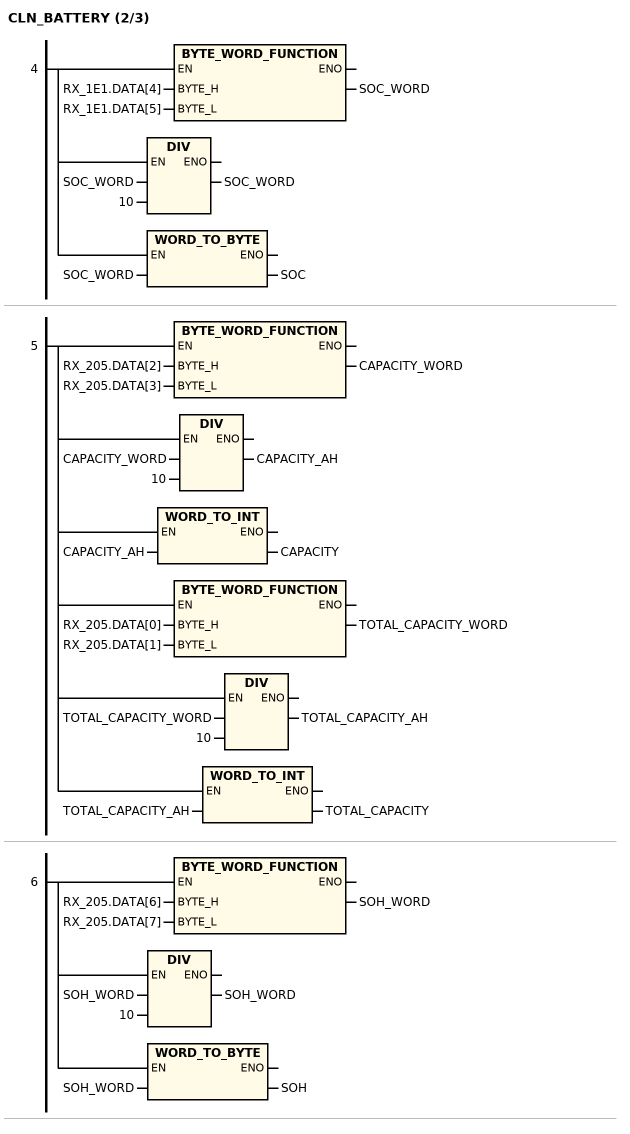
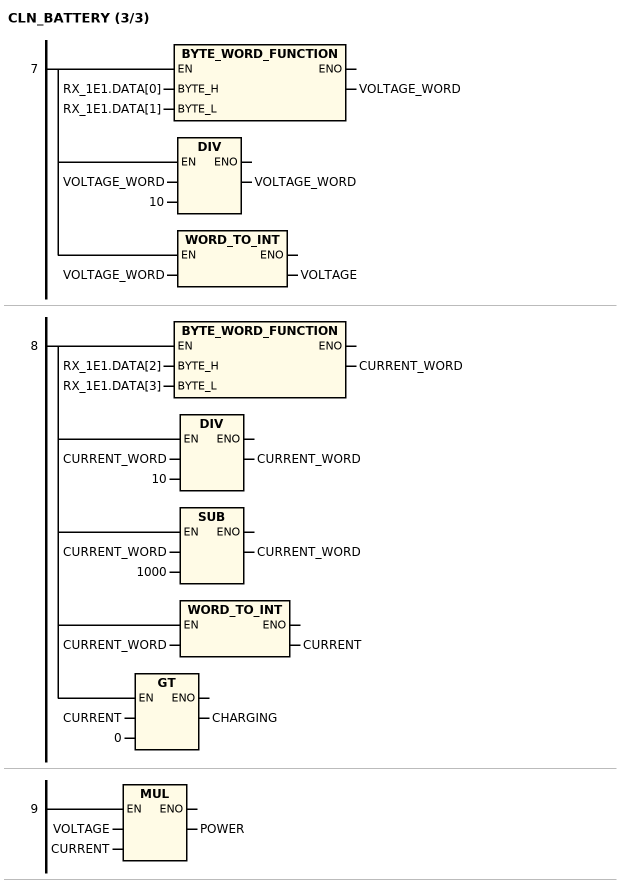
_LD_ (* Ladder Diagram *)
NETWORK 1
	*
		EN --- RX_205:RX_CAN(CHANNEL: CAN_CHANNEL, CAN_ID: 16#205)
		EN --- RX_1E1:RX_CAN(CHANNEL: CAN_CHANNEL, CAN_ID: 16#1E1)
		EN --- RX_1F5:RX_CAN(CHANNEL: CAN_CHANNEL, CAN_ID: 16#1F5)
		EN --- RX_357:RX_CAN(CHANNEL: CAN_CHANNEL, CAN_ID: 16#357)
NETWORK 2
	[RX_1E1.ERROR] - DELAY:TON(IN: *, PT: t#3s) --- (CAN_ERROR)
		EN --- MOVE(0) => SOH, SOC
		EN --- MOVE(0) => POWER, CAPACITY
		EN --- MOVE(0) => NTC_1, NTC_2
		EN --- MOVE(FALSE) => CHARGING
NETWORK 3
	*
		EN --- SUB(RX_357.DATA[2], 50) => NTC_1
		EN --- SUB(RX_357.DATA[3], 50) => NTC_2
NETWORK 4
	*
		EN --- BYTE_WORD_FUNCTION(BYTE_H: RX_1E1.DATA[4], BYTE_L: RX_1E1.DATA[5]) => SOC_WORD
		EN --- DIV(SOC_WORD, 10) => SOC_WORD
		EN --- WORD_TO_BYTE(SOC_WORD) => SOC
NETWORK 5
	*
		EN --- BYTE_WORD_FUNCTION(BYTE_H: RX_205.DATA[2], BYTE_L: RX_205.DATA[3]) => CAPACITY_WORD
		EN --- DIV(CAPACITY_WORD, 10) => CAPACITY_AH
		EN --- WORD_TO_INT(CAPACITY_AH) => CAPACITY
		EN --- BYTE_WORD_FUNCTION(BYTE_H: RX_205.DATA[0], BYTE_L: RX_205.DATA[1]) => TOTAL_CAPACITY_WORD
		EN --- DIV(TOTAL_CAPACITY_WORD, 10) => TOTAL_CAPACITY_AH
		EN --- WORD_TO_INT(TOTAL_CAPACITY_AH) => TOTAL_CAPACITY
NETWORK 6
	*
		EN --- BYTE_WORD_FUNCTION(BYTE_H: RX_205.DATA[6], BYTE_L: RX_205.DATA[7]) => SOH_WORD
		EN --- DIV(SOH_WORD, 10) => SOH_WORD
		EN --- WORD_TO_BYTE(SOH_WORD) => SOH
NETWORK 7
	*
		EN --- BYTE_WORD_FUNCTION(BYTE_H: RX_1E1.DATA[0], BYTE_L: RX_1E1.DATA[1]) => VOLTAGE_WORD
		EN --- DIV(VOLTAGE_WORD, 10) => VOLTAGE_WORD
		EN --- WORD_TO_INT(VOLTAGE_WORD) => VOLTAGE
NETWORK 8
	*
		EN --- BYTE_WORD_FUNCTION(BYTE_H: RX_1E1.DATA[2], BYTE_L: RX_1E1.DATA[3]) => CURRENT_WORD
		EN --- DIV(CURRENT_WORD, 10) => CURRENT_WORD
		EN --- SUB(CURRENT_WORD, 1000) => CURRENT_WORD
		EN --- WORD_TO_INT(CURRENT_WORD) => CURRENT
		EN --- GT(CURRENT, 0) => CHARGING
NETWORK 9
	*
		EN --- MUL(VOLTAGE, CURRENT) => POWER
_END_LD_
(* the same logic as Structured Text *)
(* Network 1 *)
RX_205(CHANNEL := CAN_CHANNEL, CAN_ID := 16#205);
RX_1E1(CHANNEL := CAN_CHANNEL, CAN_ID := 16#1E1);
RX_1F5(CHANNEL := CAN_CHANNEL, CAN_ID := 16#1F5);
RX_357(CHANNEL := CAN_CHANNEL, CAN_ID := 16#357);
(* Network 2: see the listing above *)
(* Network 3 *)
NTC_1 := RX_357.DATA[2] - 50;
NTC_2 := RX_357.DATA[3] - 50;
(* Network 4 *)
SOC_WORD := BYTE_WORD_FUNCTION(BYTE_H := RX_1E1.DATA[4], BYTE_L := RX_1E1.DATA[5]);
SOC_WORD := SOC_WORD / 10;
SOC := WORD_TO_BYTE(SOC_WORD);
(* Network 5 *)
CAPACITY_WORD := BYTE_WORD_FUNCTION(BYTE_H := RX_205.DATA[2], BYTE_L := RX_205.DATA[3]);
CAPACITY_AH := CAPACITY_WORD / 10;
CAPACITY := WORD_TO_INT(CAPACITY_AH);
TOTAL_CAPACITY_WORD := BYTE_WORD_FUNCTION(BYTE_H := RX_205.DATA[0], BYTE_L := RX_205.DATA[1]);
TOTAL_CAPACITY_AH := TOTAL_CAPACITY_WORD / 10;
TOTAL_CAPACITY := WORD_TO_INT(TOTAL_CAPACITY_AH);
(* Network 6 *)
SOH_WORD := BYTE_WORD_FUNCTION(BYTE_H := RX_205.DATA[6], BYTE_L := RX_205.DATA[7]);
SOH_WORD := SOH_WORD / 10;
SOH := WORD_TO_BYTE(SOH_WORD);
(* Network 7 *)
VOLTAGE_WORD := BYTE_WORD_FUNCTION(BYTE_H := RX_1E1.DATA[0], BYTE_L := RX_1E1.DATA[1]);
VOLTAGE_WORD := VOLTAGE_WORD / 10;
VOLTAGE := WORD_TO_INT(VOLTAGE_WORD);
(* Network 8 *)
CURRENT_WORD := BYTE_WORD_FUNCTION(BYTE_H := RX_1E1.DATA[2], BYTE_L := RX_1E1.DATA[3]);
CURRENT_WORD := CURRENT_WORD / 10;
CURRENT_WORD := CURRENT_WORD - 1000;
CURRENT := WORD_TO_INT(CURRENT_WORD);
CHARGING := CURRENT > 0;
(* Network 9 *)
POWER := VOLTAGE * CURRENT;
END_FUNCTION_BLOCK

(* POU PROGRAM_FBs/CLN_BATTERY_SELECTION, LD *)
FUNCTION_BLOCK CLN_BATTERY_SELECTION
(*
Created BY: Adiga
Date: 25-01-24
Version: 1
      
*)

VAR_INPUT
	BAT_SOC: BYTE;
	BAT_SOH: BYTE;
	BAT_POWER: INT;
	BAT_NTC1: BYTE;
	BAT_NTC2: BYTE;
	BAT_CAN_ERROR: BOOL;
	BATTERY_CAPACITY_WORD: WORD;
	BAT_CURRENT: INT;
END_VAR
VAR_OUTPUT
	LOW_SOC: BOOL;
END_VAR
VAR
	RTRIG_B1: R_TRIG;
	RTRIG_B2: R_TRIG;
	BAT_1: BOOL;
	BAT_2: BOOL;
	SOC_INT: INT;
	SOC_MAP: INT;
	SOC: BYTE;

	TON1: TON;
	TON2: TON;
END_VAR
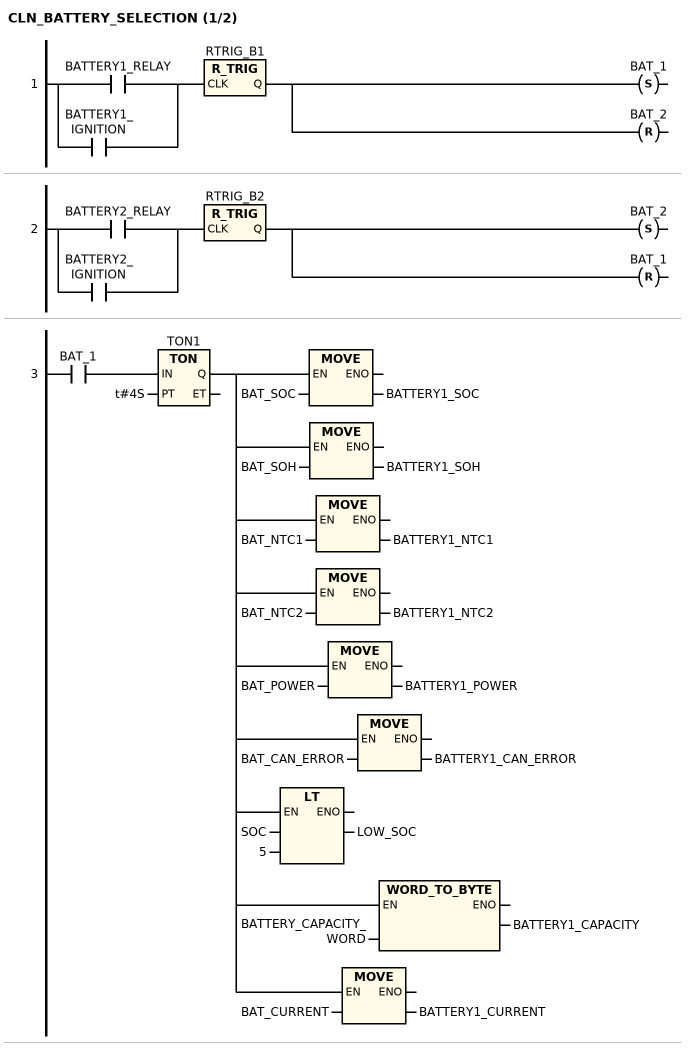
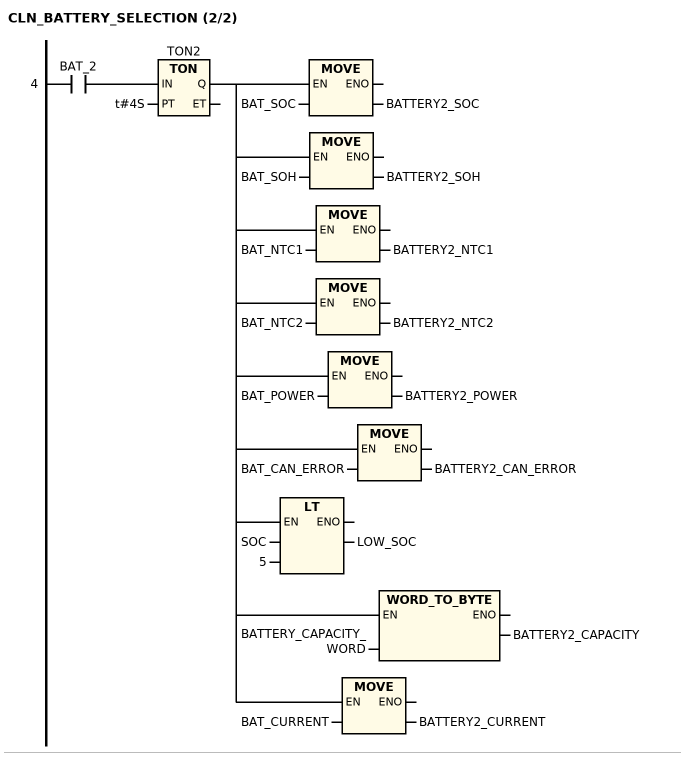
_LD_ (* Ladder Diagram *)
NETWORK 1
	{ [BATTERY1_RELAY] | [BATTERY1_IGNITION] } - RTRIG_B1:R_TRIG(CLK: *) --- (S BAT_1) (R BAT_2)
NETWORK 2
	{ [BATTERY2_RELAY] | [BATTERY2_IGNITION] } - RTRIG_B2:R_TRIG(CLK: *) --- (S BAT_2) (R BAT_1)
NETWORK 3
	[BAT_1] - TON1:TON(IN: *, PT: t#4S)
		EN --- MOVE(BAT_SOC) => BATTERY1_SOC
		EN --- MOVE(BAT_SOH) => BATTERY1_SOH
		EN --- MOVE(BAT_NTC1) => BATTERY1_NTC1
		EN --- MOVE(BAT_NTC2) => BATTERY1_NTC2
		EN --- MOVE(BAT_POWER) => BATTERY1_POWER
		EN --- MOVE(BAT_CAN_ERROR) => BATTERY1_CAN_ERROR
		EN --- LT(SOC, 5) => LOW_SOC
		EN --- WORD_TO_BYTE(BATTERY_CAPACITY_WORD) => BATTERY1_CAPACITY
		EN --- MOVE(BAT_CURRENT) => BATTERY1_CURRENT
NETWORK 4
	[BAT_2] - TON2:TON(IN: *, PT: t#4S)
		EN --- MOVE(BAT_SOC) => BATTERY2_SOC
		EN --- MOVE(BAT_SOH) => BATTERY2_SOH
		EN --- MOVE(BAT_NTC1) => BATTERY2_NTC1
		EN --- MOVE(BAT_NTC2) => BATTERY2_NTC2
		EN --- MOVE(BAT_POWER) => BATTERY2_POWER
		EN --- MOVE(BAT_CAN_ERROR) => BATTERY2_CAN_ERROR
		EN --- LT(SOC, 5) => LOW_SOC
		EN --- WORD_TO_BYTE(BATTERY_CAPACITY_WORD) => BATTERY2_CAPACITY
		EN --- MOVE(BAT_CURRENT) => BATTERY2_CURRENT
_END_LD_
(* the same logic as Structured Text *)
(* Network 1 *)
RTRIG_B1(CLK := BATTERY1_RELAY OR BATTERY1_IGNITION);
IF RTRIG_B1.Q THEN BAT_1 := TRUE; BAT_2 := FALSE; END_IF;
(* Network 2 *)
RTRIG_B2(CLK := BATTERY2_RELAY OR BATTERY2_IGNITION);
IF RTRIG_B2.Q THEN BAT_2 := TRUE; BAT_1 := FALSE; END_IF;
(* Network 3 *)
TON1(IN := BAT_1, PT := t#4S);
IF TON1.Q THEN
	BATTERY1_SOC := BAT_SOC;
	BATTERY1_SOH := BAT_SOH;
	BATTERY1_NTC1 := BAT_NTC1;
	BATTERY1_NTC2 := BAT_NTC2;
	BATTERY1_POWER := BAT_POWER;
	BATTERY1_CAN_ERROR := BAT_CAN_ERROR;
	LOW_SOC := SOC < 5;
	BATTERY1_CAPACITY := WORD_TO_BYTE(BATTERY_CAPACITY_WORD);
	BATTERY1_CURRENT := BAT_CURRENT;
END_IF;
(* Network 4 *)
TON2(IN := BAT_2, PT := t#4S);
IF TON2.Q THEN
	BATTERY2_SOC := BAT_SOC;
	BATTERY2_SOH := BAT_SOH;
	BATTERY2_NTC1 := BAT_NTC1;
	BATTERY2_NTC2 := BAT_NTC2;
	BATTERY2_POWER := BAT_POWER;
	BATTERY2_CAN_ERROR := BAT_CAN_ERROR;
	LOW_SOC := SOC < 5;
	BATTERY2_CAPACITY := WORD_TO_BYTE(BATTERY_CAPACITY_WORD);
	BATTERY2_CURRENT := BAT_CURRENT;
END_IF;
END_FUNCTION_BLOCK

(* POU PROGRAM_FBs/CLN_BATTERY_SELECTION_2, LD *)
 FUNCTION_BLOCK CLN_BATTERY_SELECTION_2
VAR_INPUT
	BAT_SOC: BYTE;
	BAT_SOH: BYTE;
	BAT_POWER: INT;
	BAT_NTC1: BYTE;
	BAT_NTC2: BYTE;
	BAT_CAN_ERROR: BOOL;
	BAT_CURRENT: INT;
END_VAR
VAR_OUTPUT
END_VAR
VAR
	BAT1_TON: TON;
	BAT2_TON: TON;
END_VAR
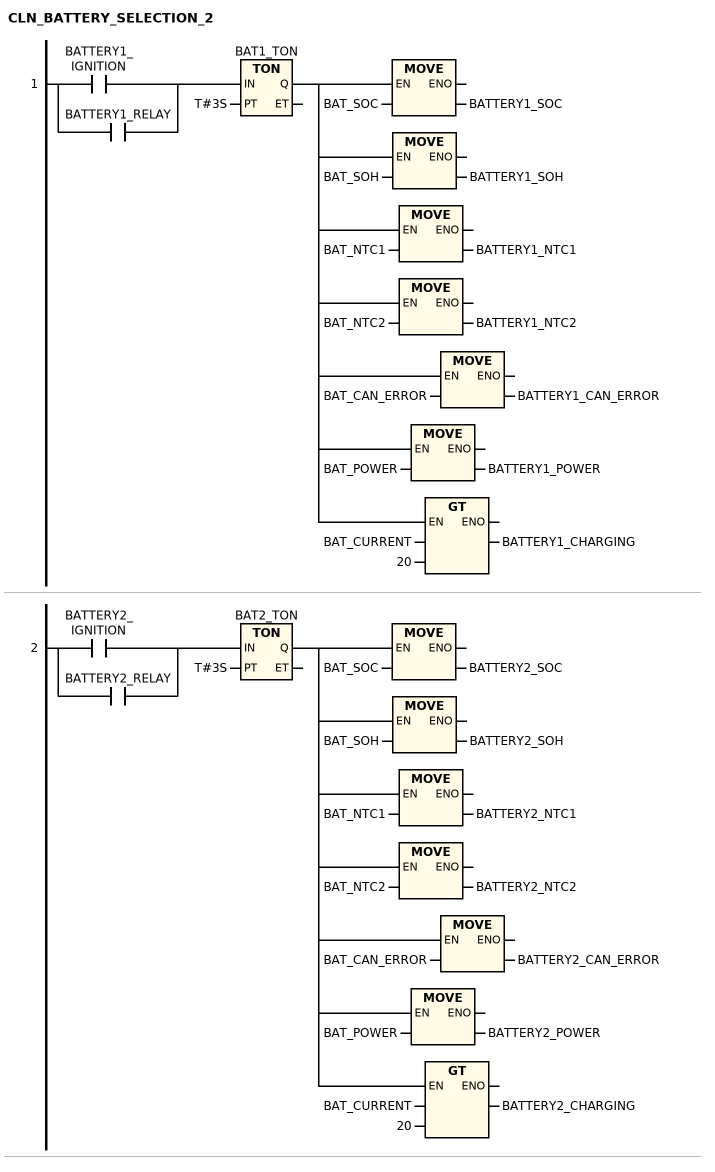
_LD_ (* Ladder Diagram *)
NETWORK 1
	{ [BATTERY1_IGNITION] | [BATTERY1_RELAY] } - BAT1_TON:TON(IN: *, PT: T#3S)
		EN --- MOVE(BAT_SOC) => BATTERY1_SOC
		EN --- MOVE(BAT_SOH) => BATTERY1_SOH
		EN --- MOVE(BAT_NTC1) => BATTERY1_NTC1
		EN --- MOVE(BAT_NTC2) => BATTERY1_NTC2
		EN --- MOVE(BAT_CAN_ERROR) => BATTERY1_CAN_ERROR
		EN --- MOVE(BAT_POWER) => BATTERY1_POWER
		EN --- GT(BAT_CURRENT, 20) => BATTERY1_CHARGING
NETWORK 2
	{ [BATTERY2_IGNITION] | [BATTERY2_RELAY] } - BAT2_TON:TON(IN: *, PT: T#3S)
		EN --- MOVE(BAT_SOC) => BATTERY2_SOC
		EN --- MOVE(BAT_SOH) => BATTERY2_SOH
		EN --- MOVE(BAT_NTC1) => BATTERY2_NTC1
		EN --- MOVE(BAT_NTC2) => BATTERY2_NTC2
		EN --- MOVE(BAT_CAN_ERROR) => BATTERY2_CAN_ERROR
		EN --- MOVE(BAT_POWER) => BATTERY2_POWER
		EN --- GT(BAT_CURRENT, 20) => BATTERY2_CHARGING
_END_LD_
(* the same logic as Structured Text *)
(* Network 1 *)
BAT1_TON(IN := BATTERY1_IGNITION OR BATTERY1_RELAY, PT := T#3S);
IF BAT1_TON.Q THEN
	BATTERY1_SOC := BAT_SOC;
	BATTERY1_SOH := BAT_SOH;
	BATTERY1_NTC1 := BAT_NTC1;
	BATTERY1_NTC2 := BAT_NTC2;
	BATTERY1_CAN_ERROR := BAT_CAN_ERROR;
	BATTERY1_POWER := BAT_POWER;
	BATTERY1_CHARGING := BAT_CURRENT > 20;
END_IF;
(* Network 2 *)
BAT2_TON(IN := BATTERY2_IGNITION OR BATTERY2_RELAY, PT := T#3S);
IF BAT2_TON.Q THEN
	BATTERY2_SOC := BAT_SOC;
	BATTERY2_SOH := BAT_SOH;
	BATTERY2_NTC1 := BAT_NTC1;
	BATTERY2_NTC2 := BAT_NTC2;
	BATTERY2_CAN_ERROR := BAT_CAN_ERROR;
	BATTERY2_POWER := BAT_POWER;
	BATTERY2_CHARGING := BAT_CURRENT > 20;
END_IF;
END_FUNCTION_BLOCK

(* POU PROGRAM_FBs/CLN_BATTERY_SWITCH, LD *)
FUNCTION_BLOCK CLN_BATTERY_SWITCH

(*THIS BLOCK IS COMPATIBLE FOR 2X CLN BATTERIES*)

VAR_INPUT
	CHARGER_IN: BOOL;
	IGN_KEY: BOOL;
	BAT1_IGNITION: BOOL;
	BAT2_IGNITION: BOOL;
	SOC_BAT1: BYTE;
	SOC_BAT2: BYTE;
	BAT1_CAN_ERROR: BOOL;
	BAT2_CAN_ERROR: BOOL;
END_VAR

VAR_OUTPUT
	RELAY_BAT1: BOOL;
	RELAY_BAT2: BOOL;
	ERROR: BOOL;
END_VAR

VAR
	BAT1_CAN_TIMER: TON;
	BAT2_CAN_TIMER: TON;
	BAT1_FULL: BOOL;
	BAT2_FULL: BOOL;
	BAT1_80: BOOL;
	BAT2_80: BOOL;
	CHARGE_1: BOOL;
	RELAY1_TIMER: TON;
	RELAY2_TIMER: TON;
	BLUE_BLINK: BLINK;
	CHARGE1_BLINK: BLINK;
	CHARGE2_BLINK: BLINK;
	CHARGING_SAFETY: BOOL;

	ERROR_TIMER: TON;
END_VAR
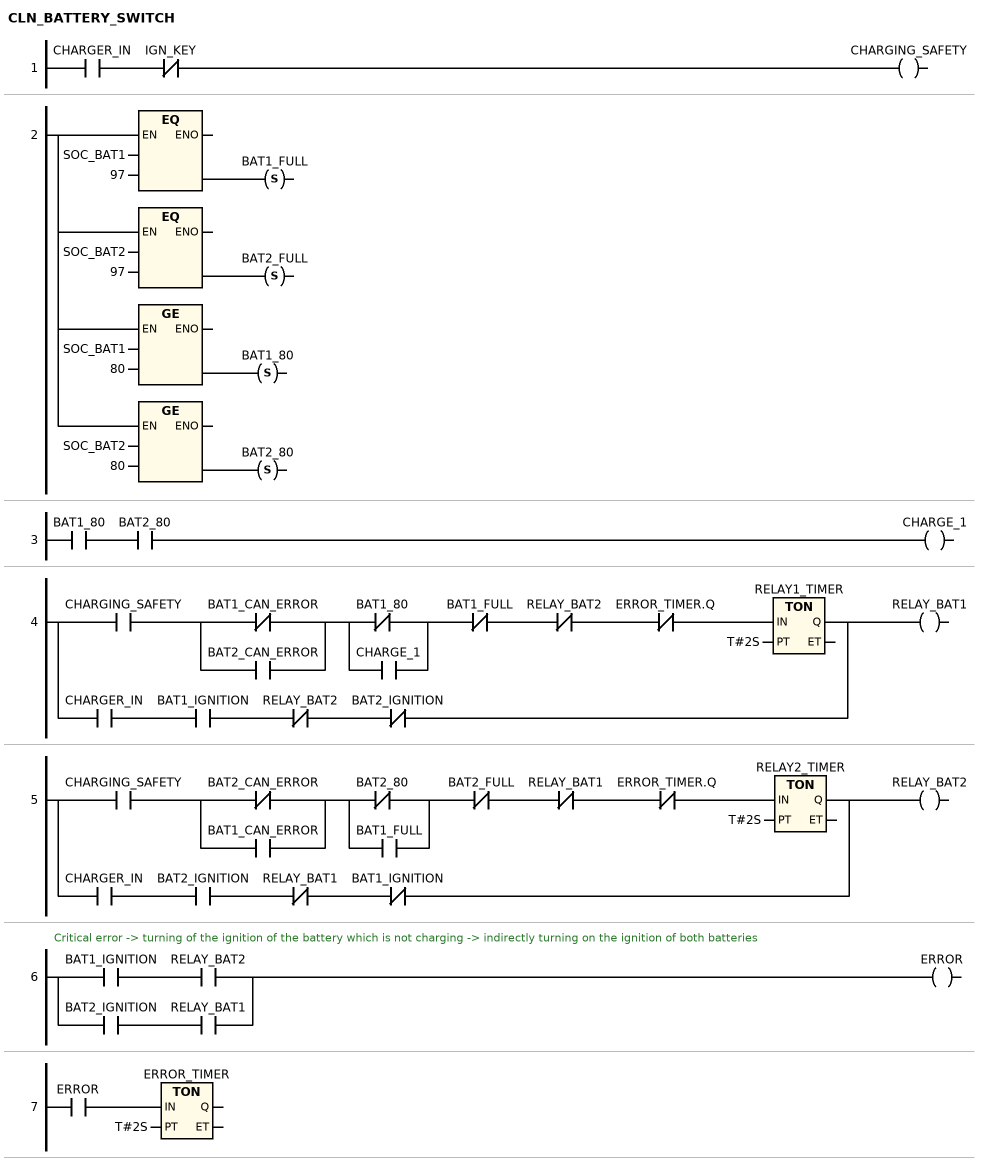
_LD_ (* Ladder Diagram *)
NETWORK 1
	[CHARGER_IN] - [/IGN_KEY] --- (CHARGING_SAFETY)
NETWORK 2
	*
		EN --- EQ(SOC_BAT1, 97) => S BAT1_FULL
		EN --- EQ(SOC_BAT2, 97) => S BAT2_FULL
		EN --- GE(SOC_BAT1, 80) => S BAT1_80
		EN --- GE(SOC_BAT2, 80) => S BAT2_80
NETWORK 3
	[BAT1_80] - [BAT2_80] --- (CHARGE_1)
NETWORK 4
	{ [CHARGING_SAFETY] - { [/BAT1_CAN_ERROR] | [BAT2_CAN_ERROR] } - { [/BAT1_80] | [CHARGE_1] } - [/BAT1_FULL] - [/RELAY_BAT2] - [/ERROR_TIMER.Q] - RELAY1_TIMER:TON(IN: *, PT: T#2S) | [CHARGER_IN] - [BAT1_IGNITION] - [/RELAY_BAT2] - [/BAT2_IGNITION] } --- (RELAY_BAT1)
NETWORK 5
	{ [CHARGING_SAFETY] - { [/BAT2_CAN_ERROR] | [BAT1_CAN_ERROR] } - { [/BAT2_80] | [BAT1_FULL] } - [/BAT2_FULL] - [/RELAY_BAT1] - [/ERROR_TIMER.Q] - RELAY2_TIMER:TON(IN: *, PT: T#2S) | [CHARGER_IN] - [BAT2_IGNITION] - [/RELAY_BAT1] - [/BAT1_IGNITION] } --- (RELAY_BAT2)
NETWORK 6 (* Critical error -> turning of the ignition of the battery which is not charging -> indirectly turning on the ignition of both batteries *)
	{ [BAT1_IGNITION] - [RELAY_BAT2] | [BAT2_IGNITION] - [RELAY_BAT1] } --- (ERROR)
NETWORK 7
	[ERROR] - ERROR_TIMER:TON(IN: *, PT: T#2S)
_END_LD_
(* the same logic as Structured Text *)
(* Network 1 *)
CHARGING_SAFETY := CHARGER_IN AND NOT IGN_KEY;
(* Network 2 *)
IF SOC_BAT1 = 97 THEN BAT1_FULL := TRUE; END_IF;
IF SOC_BAT2 = 97 THEN BAT2_FULL := TRUE; END_IF;
IF SOC_BAT1 >= 80 THEN BAT1_80 := TRUE; END_IF;
IF SOC_BAT2 >= 80 THEN BAT2_80 := TRUE; END_IF;
(* Network 3 *)
CHARGE_1 := BAT1_80 AND BAT2_80;
(* Network 4 *)
RELAY1_TIMER(IN := CHARGING_SAFETY AND (NOT BAT1_CAN_ERROR OR BAT2_CAN_ERROR) AND (NOT BAT1_80 OR CHARGE_1) AND NOT BAT1_FULL AND NOT RELAY_BAT2 AND NOT ERROR_TIMER.Q, PT := T#2S);
RELAY_BAT1 := RELAY1_TIMER.Q OR CHARGER_IN AND BAT1_IGNITION AND NOT RELAY_BAT2 AND NOT BAT2_IGNITION;
(* Network 5 *)
RELAY2_TIMER(IN := CHARGING_SAFETY AND (NOT BAT2_CAN_ERROR OR BAT1_CAN_ERROR) AND (NOT BAT2_80 OR BAT1_FULL) AND NOT BAT2_FULL AND NOT RELAY_BAT1 AND NOT ERROR_TIMER.Q, PT := T#2S);
RELAY_BAT2 := RELAY2_TIMER.Q OR CHARGER_IN AND BAT2_IGNITION AND NOT RELAY_BAT1 AND NOT BAT1_IGNITION;
(* Network 6: Critical error -> turning of the ignition of the battery which is not charging -> indirectly turning on the ignition of both batteries *)
ERROR := BAT1_IGNITION AND RELAY_BAT2 OR BAT2_IGNITION AND RELAY_BAT1;
(* Network 7 *)
ERROR_TIMER(IN := ERROR, PT := T#2S);
END_FUNCTION_BLOCK

(* POU PROGRAM_FBs/CLN_CHARGING, LD *)
FUNCTION_BLOCK CLN_CHARGING
(*
THIS BLOCK IS COMPATIBLE FOR 2X CLN BATTERIES0

Created BY: Adiga
Date: 25-01-24
UPDATED :14-03-25
Version: 4
1.DUAL BATTERY CAHRGING BLOCK ONLY FOR CLN
2.UPDATED THE BLOCK FOR CHARGING WITH AND WITHOUT IGN ON
3.ADDED BATTERY CAN ERROR CODITION TO CHARGE
4.ADDED TIMER BEFORE SWITCHING BATTRY BELAY.
.
*)

VAR_INPUT
	CHANNEL: BYTE;
	CHARGER_IN: BOOL;
	IGN_KEY: BOOL;
	BAT1_IGN: BOOL;
	BAT2_IGN: BOOL;
	SOC1: BYTE;
	SOC2: BYTE;
	BAT_CAN_ERROR1: BOOL;
	BAT_CAN_ERROR2: BOOL;
	BATTERY_CHARGING: BOOL;
END_VAR

VAR_OUTPUT
	RELAY_BAT1: BOOL;
	RELAY_BAT2: BOOL;
	BLUE_LED_OUT: BOOL;
	ERROR: BOOL;
	BUZZER_ON: BOOL;
	CHARGING1: BOOL;
	CHARGING2: BOOL;
END_VAR

VAR
	CHARGE_1: BOOL;
	BAT_1_FULL: BOOL;
	BAT_2_FULL: BOOL;
	T1: TON;
	T2: TON;
	T3: TON;
	IGNITION_OFF: BOOL;
	BAT_1_80: BOOL;
	BAT_2_80: BOOL;
	FTRIG1: F_TRIG;
	TIMER5: TON;
	T4: TON;
	T5: TON;
	CHARGING_2: BLINK;
	CHARGING_1: BLINK;
END_VAR
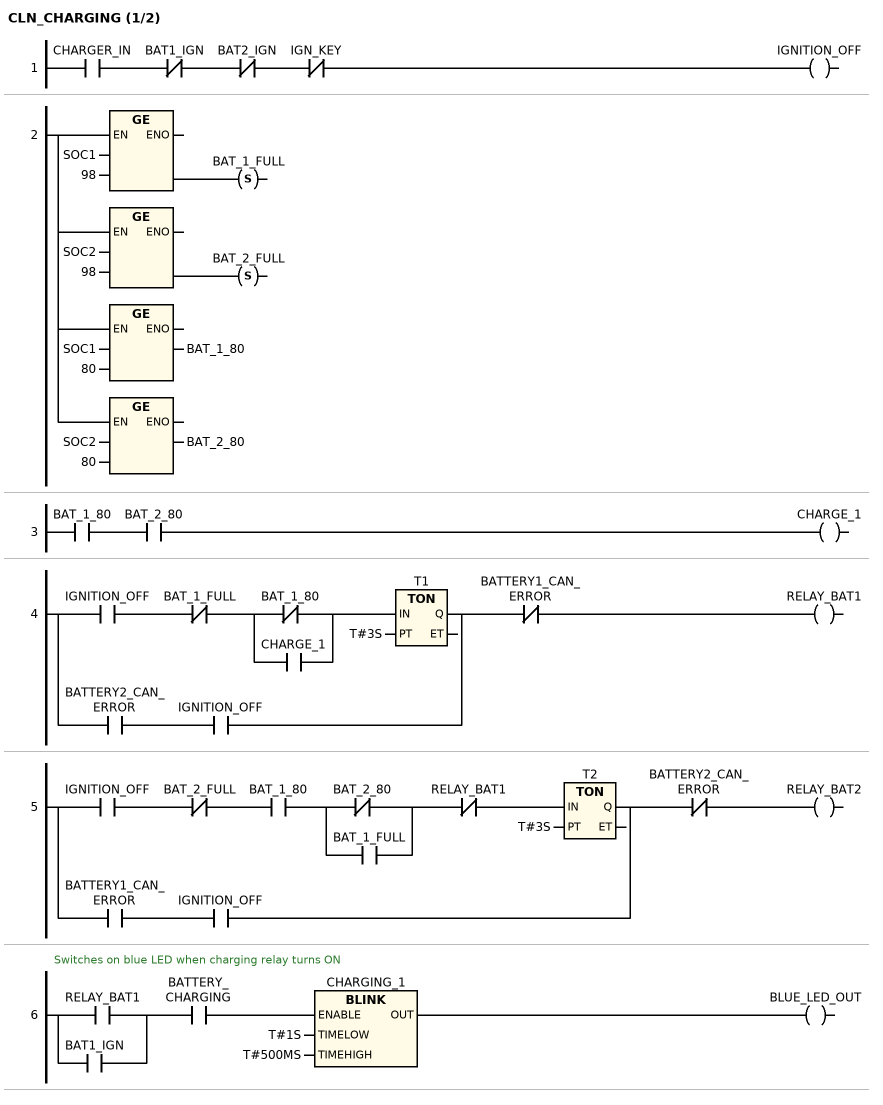
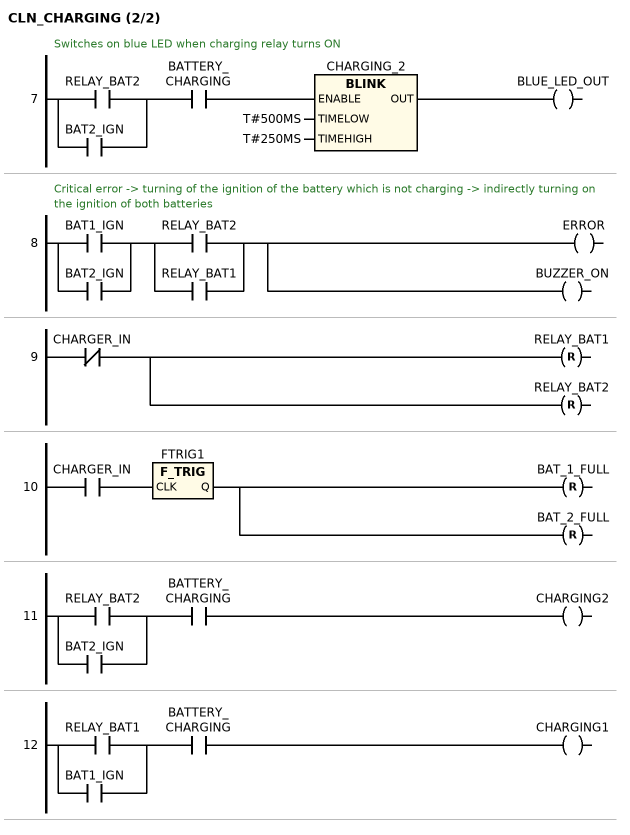
_LD_ (* Ladder Diagram *)
NETWORK 1
	[CHARGER_IN] - [/BAT1_IGN] - [/BAT2_IGN] - [/IGN_KEY] --- (IGNITION_OFF)
NETWORK 2
	*
		EN --- GE(SOC1, 98) => S BAT_1_FULL
		EN --- GE(SOC2, 98) => S BAT_2_FULL
		EN --- GE(SOC1, 80) => BAT_1_80
		EN --- GE(SOC2, 80) => BAT_2_80
NETWORK 3
	[BAT_1_80] - [BAT_2_80] --- (CHARGE_1)
NETWORK 4
	{ [IGNITION_OFF] - [/BAT_1_FULL] - { [/BAT_1_80] | [CHARGE_1] } - T1:TON(IN: *, PT: T#3S) | [BATTERY2_CAN_ERROR] - [IGNITION_OFF] } - [/BATTERY1_CAN_ERROR] --- (RELAY_BAT1)
NETWORK 5
	{ [IGNITION_OFF] - [/BAT_2_FULL] - [BAT_1_80] - { [/BAT_2_80] | [BAT_1_FULL] } - [/RELAY_BAT1] - T2:TON(IN: *, PT: T#3S) | [BATTERY1_CAN_ERROR] - [IGNITION_OFF] } - [/BATTERY2_CAN_ERROR] --- (RELAY_BAT2)
NETWORK 6 (* Switches on blue LED when charging relay turns ON *)
	{ [RELAY_BAT1] | [BAT1_IGN] } - [BATTERY_CHARGING] - CHARGING_1:BLINK(ENABLE: *, TIMELOW: T#1S, TIMEHIGH: T#500MS) --- (BLUE_LED_OUT)
NETWORK 7 (* Switches on blue LED when charging relay turns ON *)
	{ [RELAY_BAT2] | [BAT2_IGN] } - [BATTERY_CHARGING] - CHARGING_2:BLINK(ENABLE: *, TIMELOW: T#500MS, TIMEHIGH: T#250MS) --- (BLUE_LED_OUT)
NETWORK 8 (* Critical error -> turning of the ignition of the battery which is not charging -> indirectly turning on the ignition of both batteries *)
	{ [BAT1_IGN] | [BAT2_IGN] } - { [RELAY_BAT2] | [RELAY_BAT1] } --- (ERROR) (BUZZER_ON)
NETWORK 9
	[/CHARGER_IN] --- (R RELAY_BAT1) (R RELAY_BAT2)
NETWORK 10
	[CHARGER_IN] - FTRIG1:F_TRIG(CLK: *) --- (R BAT_1_FULL) (R BAT_2_FULL)
NETWORK 11
	{ [RELAY_BAT2] | [BAT2_IGN] } - [BATTERY_CHARGING] --- (CHARGING2)
NETWORK 12
	{ [RELAY_BAT1] | [BAT1_IGN] } - [BATTERY_CHARGING] --- (CHARGING1)
_END_LD_
(* the same logic as Structured Text *)
(* Network 1 *)
IGNITION_OFF := CHARGER_IN AND NOT BAT1_IGN AND NOT BAT2_IGN AND NOT IGN_KEY;
(* Network 2 *)
IF SOC1 >= 98 THEN BAT_1_FULL := TRUE; END_IF;
IF SOC2 >= 98 THEN BAT_2_FULL := TRUE; END_IF;
BAT_1_80 := SOC1 >= 80;
BAT_2_80 := SOC2 >= 80;
(* Network 3 *)
CHARGE_1 := BAT_1_80 AND BAT_2_80;
(* Network 4 *)
T1(IN := IGNITION_OFF AND NOT BAT_1_FULL AND (NOT BAT_1_80 OR CHARGE_1), PT := T#3S);
RELAY_BAT1 := (T1.Q OR BATTERY2_CAN_ERROR AND IGNITION_OFF) AND NOT BATTERY1_CAN_ERROR;
(* Network 5 *)
T2(IN := IGNITION_OFF AND NOT BAT_2_FULL AND BAT_1_80 AND (NOT BAT_2_80 OR BAT_1_FULL) AND NOT RELAY_BAT1, PT := T#3S);
RELAY_BAT2 := (T2.Q OR BATTERY1_CAN_ERROR AND IGNITION_OFF) AND NOT BATTERY2_CAN_ERROR;
(* Network 6: Switches on blue LED when charging relay turns ON *)
CHARGING_1(ENABLE := (RELAY_BAT1 OR BAT1_IGN) AND BATTERY_CHARGING, TIMELOW := T#1S, TIMEHIGH := T#500MS);
BLUE_LED_OUT := CHARGING_1.OUT;
(* Network 7: Switches on blue LED when charging relay turns ON *)
CHARGING_2(ENABLE := (RELAY_BAT2 OR BAT2_IGN) AND BATTERY_CHARGING, TIMELOW := T#500MS, TIMEHIGH := T#250MS);
BLUE_LED_OUT := CHARGING_2.OUT;
(* Network 8: Critical error -> turning of the ignition of the battery which is not charging -> indirectly turning on the ignition of both batteries *)
ERROR := (BAT1_IGN OR BAT2_IGN) AND (RELAY_BAT2 OR RELAY_BAT1);
BUZZER_ON := ERROR;
(* Network 9 *)
IF NOT CHARGER_IN THEN RELAY_BAT1 := FALSE; RELAY_BAT2 := FALSE; END_IF;
(* Network 10 *)
FTRIG1(CLK := CHARGER_IN);
IF FTRIG1.Q THEN BAT_1_FULL := FALSE; BAT_2_FULL := FALSE; END_IF;
(* Network 11 *)
CHARGING2 := (RELAY_BAT2 OR BAT2_IGN) AND BATTERY_CHARGING;
(* Network 12 *)
CHARGING1 := (RELAY_BAT1 OR BAT1_IGN) AND BATTERY_CHARGING;
END_FUNCTION_BLOCK

(* POU PROGRAM_FBs/DRIVE_LOGIC, LD *)
FUNCTION_BLOCK DRIVE_LOGIC
VAR_INPUT
	JX: INT;
	JY: INT;
	LEFT_BUTTON: BOOL;
	JOY_ORIGIN: BOOL;
	EM_SWITCH_IN: BOOL;
	OVER_TEMP: BOOL;
END_VAR
VAR_OUTPUT
	JX_1: INT;
	JY_1: INT;
	DISARM: BOOL;
	EM_BRAKE_OUT: BOOL;
	DRIVE_ERROR: BOOL;
END_VAR
VAR
	SLEEP_TIMER: TON;
	ON_DELAY: TON;
	APPLY_EM: BOOL;
	LOW_RPM: BOOL;
	EMFB_ERROR: BOOL;
END_VAR
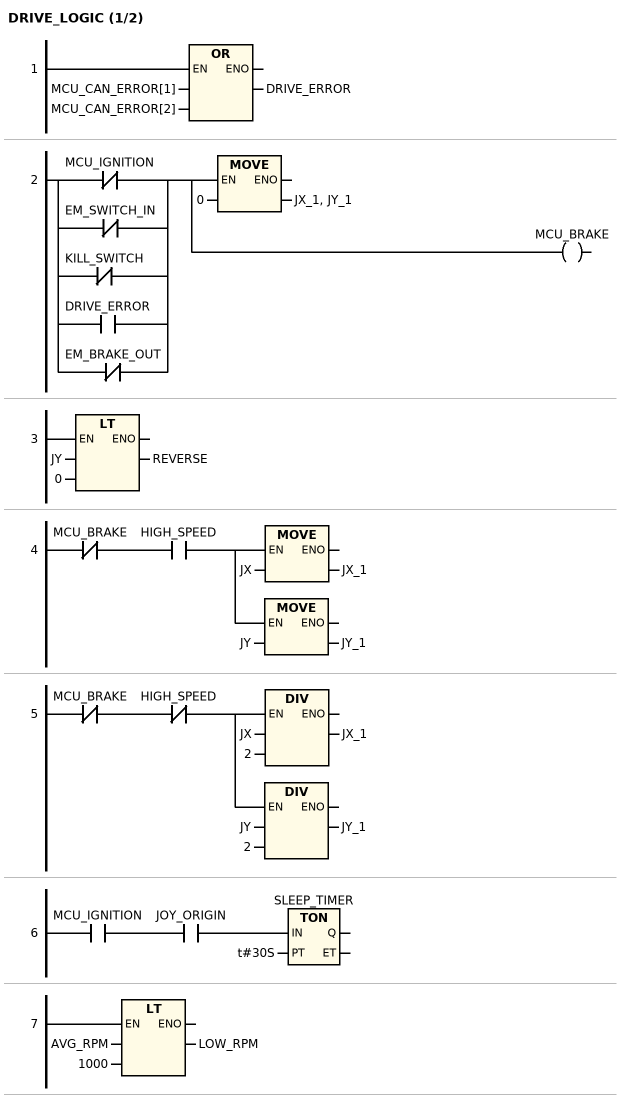
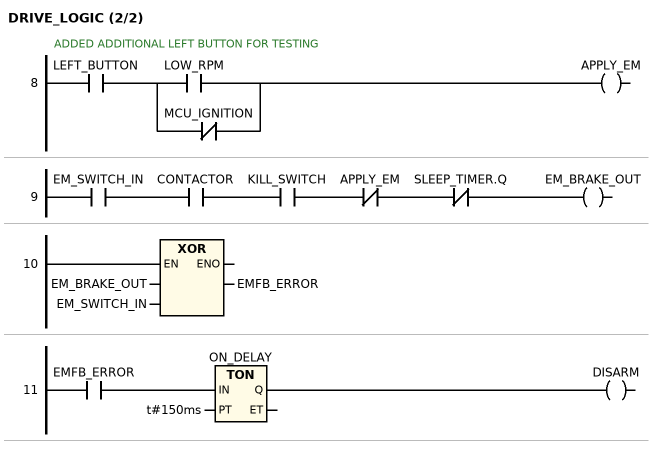
_LD_ (* Ladder Diagram *)
NETWORK 1
	*
		EN --- OR(MCU_CAN_ERROR[1], MCU_CAN_ERROR[2]) => DRIVE_ERROR
NETWORK 2
	{ [/MCU_IGNITION] | [/EM_SWITCH_IN] | [/KILL_SWITCH] | [DRIVE_ERROR] | [/EM_BRAKE_OUT] } --- (MCU_BRAKE)
		EN --- MOVE(0) => JX_1, JY_1
NETWORK 3
	*
		EN --- LT(JY, 0) => REVERSE
NETWORK 4
	[/MCU_BRAKE] - [HIGH_SPEED]
		EN --- MOVE(JX) => JX_1
		EN --- MOVE(JY) => JY_1
NETWORK 5
	[/MCU_BRAKE] - [/HIGH_SPEED]
		EN --- DIV(JX, 2) => JX_1
		EN --- DIV(JY, 2) => JY_1
NETWORK 6
	[MCU_IGNITION] - [JOY_ORIGIN] - SLEEP_TIMER:TON(IN: *, PT: t#30S)
NETWORK 7
	*
		EN --- LT(AVG_RPM, 1000) => LOW_RPM
NETWORK 8 (* ADDED ADDITIONAL LEFT BUTTON FOR TESTING *)
	[LEFT_BUTTON] - { [LOW_RPM] | [/MCU_IGNITION] } --- (APPLY_EM)
NETWORK 9
	[EM_SWITCH_IN] - [CONTACTOR] - [KILL_SWITCH] - [/APPLY_EM] - [/SLEEP_TIMER.Q] --- (EM_BRAKE_OUT)
NETWORK 10
	*
		EN --- XOR(EM_BRAKE_OUT, EM_SWITCH_IN) => EMFB_ERROR
NETWORK 11
	[EMFB_ERROR] - ON_DELAY:TON(IN: *, PT: t#150ms) --- (DISARM)
_END_LD_
(* the same logic as Structured Text *)
(* Network 1 *)
DRIVE_ERROR := MCU_CAN_ERROR[1] OR MCU_CAN_ERROR[2];
(* Network 2: see the listing above *)
(* Network 3 *)
REVERSE := JY < 0;
(* Network 4 *)
IF NOT MCU_BRAKE AND HIGH_SPEED THEN
	JX_1 := JX;
	JY_1 := JY;
END_IF;
(* Network 5 *)
IF NOT MCU_BRAKE AND NOT HIGH_SPEED THEN
	JX_1 := JX / 2;
	JY_1 := JY / 2;
END_IF;
(* Network 6 *)
SLEEP_TIMER(IN := MCU_IGNITION AND JOY_ORIGIN, PT := t#30S);
(* Network 7 *)
LOW_RPM := AVG_RPM < 1000;
(* Network 8 *)
APPLY_EM := LEFT_BUTTON AND (LOW_RPM OR NOT MCU_IGNITION);
(* Network 9 *)
EM_BRAKE_OUT := EM_SWITCH_IN AND CONTACTOR AND KILL_SWITCH AND NOT APPLY_EM AND NOT SLEEP_TIMER.Q;
(* Network 10 *)
EMFB_ERROR := EM_BRAKE_OUT XOR EM_SWITCH_IN;
(* Network 11 *)
ON_DELAY(IN := EMFB_ERROR, PT := t#150ms);
DISARM := ON_DELAY.Q;
END_FUNCTION_BLOCK

(* POU PROGRAM_FBs/DUAL_CLN_CHARGING, LD *)
FUNCTION_BLOCK DUAL_CLN_CHARGING
(*
THIS BLOCK IS COMPATIBLE FOR 2X CLN BATTERIES

Created BY: Adiga
Date: 8-08-24
Version: 1
 
*)

VAR_INPUT
	CHANNEL: BYTE;
	CHARGER_IN: BOOL;
	BAT_CAN_ERROR1: BOOL;
	BAT_CAN_ERROR2: BOOL;
	BAT1_IGN: BOOL;
	BAT2_IGN: BOOL;
	BATTERY_CHARGING: BOOL;

END_VAR

VAR_OUTPUT
	RELAY_BAT1: BOOL;
	RELAY_BAT2: BOOL;
	BLUE_LED_OUT: BOOL;
	ERROR: BOOL;
	BUZZER_ON: BOOL;
	CHARGING1: BOOL;
	CHARGING2: BOOL;
END_VAR

VAR
	CHARGE_1: BOOL;
	BAT_1_FULL: BOOL;
	BAT_2_FULL: BOOL;
	RX_SOLTERRA: RX_CAN;
	CHARGER_TIMER: TON;
	SOLTERRA_TX: CAN_TX;
	CHARGING_FRAME: ARRAY [0..7] OF BYTE  := 16#03,16#25,16#01,16#5E,0,0,0,0;

	T1: TON;
	T2: TON;
	T3: TON;
	SOC2: BYTE;
	SOC1: BYTE;
	TX_CLN: CAN_TX;
	IGNITION_OFF: BOOL;
	BAT_1_80: BOOL;
	BAT_2_80: BOOL;
	FTRIG1: F_TRIG;
	TIMER5: TON;
	T4: TON;
	T5: TON;

	CHARGE: F_TRIG;
END_VAR
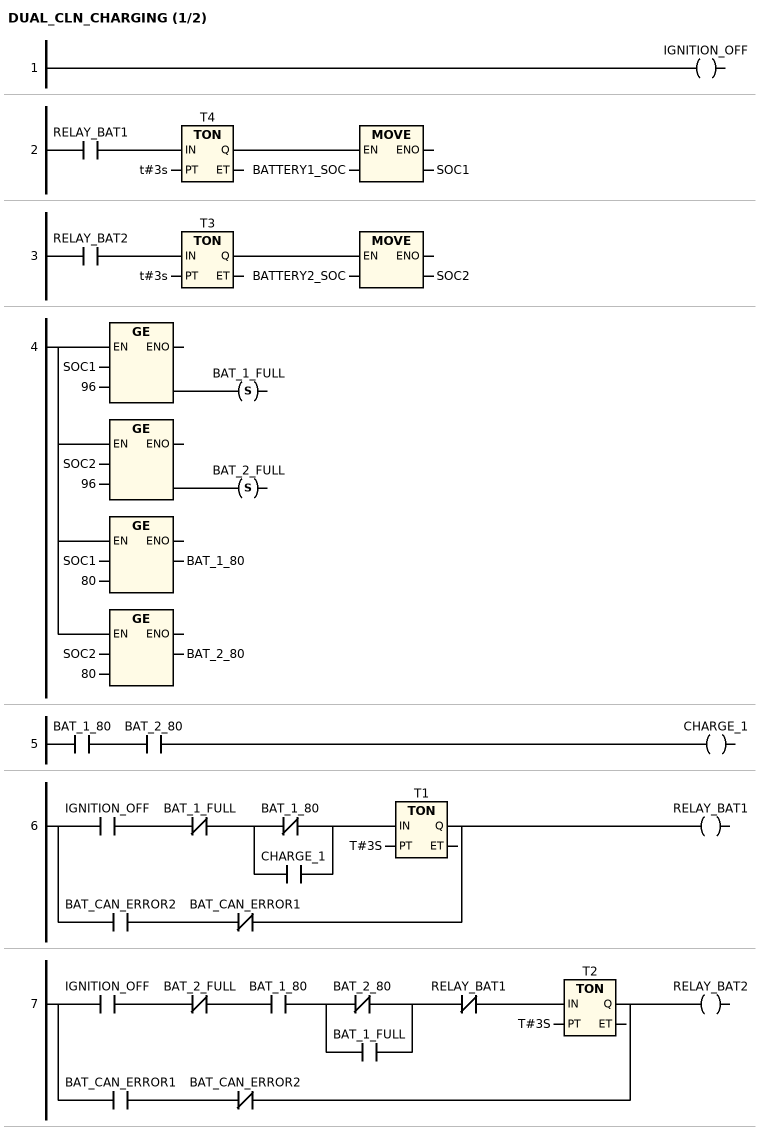
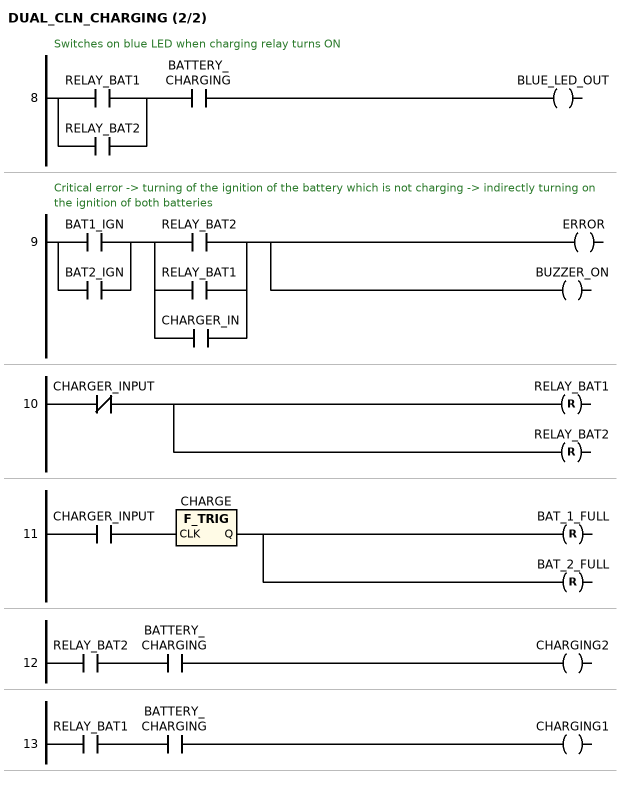
_LD_ (* Ladder Diagram *)
NETWORK 1
	* --- (IGNITION_OFF)
NETWORK 2
	[RELAY_BAT1] - T4:TON(IN: *, PT: t#3s)
		EN --- MOVE(BATTERY1_SOC) => SOC1
NETWORK 3
	[RELAY_BAT2] - T3:TON(IN: *, PT: t#3s)
		EN --- MOVE(BATTERY2_SOC) => SOC2
NETWORK 4
	*
		EN --- GE(SOC1, 96) => S BAT_1_FULL
		EN --- GE(SOC2, 96) => S BAT_2_FULL
		EN --- GE(SOC1, 80) => BAT_1_80
		EN --- GE(SOC2, 80) => BAT_2_80
NETWORK 5
	[BAT_1_80] - [BAT_2_80] --- (CHARGE_1)
NETWORK 6
	{ [IGNITION_OFF] - [/BAT_1_FULL] - { [/BAT_1_80] | [CHARGE_1] } - T1:TON(IN: *, PT: T#3S) | [BAT_CAN_ERROR2] - [/BAT_CAN_ERROR1] } --- (RELAY_BAT1)
NETWORK 7
	{ [IGNITION_OFF] - [/BAT_2_FULL] - [BAT_1_80] - { [/BAT_2_80] | [BAT_1_FULL] } - [/RELAY_BAT1] - T2:TON(IN: *, PT: T#3S) | [BAT_CAN_ERROR1] - [/BAT_CAN_ERROR2] } --- (RELAY_BAT2)
NETWORK 8 (* Switches on blue LED when charging relay turns ON *)
	{ [RELAY_BAT1] | [RELAY_BAT2] } - [BATTERY_CHARGING] --- (BLUE_LED_OUT)
NETWORK 9 (* Critical error -> turning of the ignition of the battery which is not charging -> indirectly turning on the ignition of both batteries *)
	{ [BAT1_IGN] | [BAT2_IGN] } - { [RELAY_BAT2] | [RELAY_BAT1] | [CHARGER_IN] } --- (ERROR) (BUZZER_ON)
NETWORK 10
	[/CHARGER_INPUT] --- (R RELAY_BAT1) (R RELAY_BAT2)
NETWORK 11
	[CHARGER_INPUT] - CHARGE:F_TRIG(CLK: *) --- (R BAT_1_FULL) (R BAT_2_FULL)
NETWORK 12
	[RELAY_BAT2] - [BATTERY_CHARGING] --- (CHARGING2)
NETWORK 13
	[RELAY_BAT1] - [BATTERY_CHARGING] --- (CHARGING1)
_END_LD_
(* the same logic as Structured Text *)
(* Network 1 *)
IGNITION_OFF := TRUE;
(* Network 2 *)
T4(IN := RELAY_BAT1, PT := t#3s);
IF T4.Q THEN
	SOC1 := BATTERY1_SOC;
END_IF;
(* Network 3 *)
T3(IN := RELAY_BAT2, PT := t#3s);
IF T3.Q THEN
	SOC2 := BATTERY2_SOC;
END_IF;
(* Network 4 *)
IF SOC1 >= 96 THEN BAT_1_FULL := TRUE; END_IF;
IF SOC2 >= 96 THEN BAT_2_FULL := TRUE; END_IF;
BAT_1_80 := SOC1 >= 80;
BAT_2_80 := SOC2 >= 80;
(* Network 5 *)
CHARGE_1 := BAT_1_80 AND BAT_2_80;
(* Network 6 *)
T1(IN := IGNITION_OFF AND NOT BAT_1_FULL AND (NOT BAT_1_80 OR CHARGE_1), PT := T#3S);
RELAY_BAT1 := T1.Q OR BAT_CAN_ERROR2 AND NOT BAT_CAN_ERROR1;
(* Network 7 *)
T2(IN := IGNITION_OFF AND NOT BAT_2_FULL AND BAT_1_80 AND (NOT BAT_2_80 OR BAT_1_FULL) AND NOT RELAY_BAT1, PT := T#3S);
RELAY_BAT2 := T2.Q OR BAT_CAN_ERROR1 AND NOT BAT_CAN_ERROR2;
(* Network 8: Switches on blue LED when charging relay turns ON *)
BLUE_LED_OUT := (RELAY_BAT1 OR RELAY_BAT2) AND BATTERY_CHARGING;
(* Network 9: Critical error -> turning of the ignition of the battery which is not charging -> indirectly turning on the ignition of both batteries *)
ERROR := (BAT1_IGN OR BAT2_IGN) AND (RELAY_BAT2 OR RELAY_BAT1 OR CHARGER_IN);
BUZZER_ON := ERROR;
(* Network 10 *)
IF NOT CHARGER_INPUT THEN RELAY_BAT1 := FALSE; RELAY_BAT2 := FALSE; END_IF;
(* Network 11 *)
CHARGE(CLK := CHARGER_INPUT);
IF CHARGE.Q THEN BAT_1_FULL := FALSE; BAT_2_FULL := FALSE; END_IF;
(* Network 12 *)
CHARGING2 := RELAY_BAT2 AND BATTERY_CHARGING;
(* Network 13 *)
CHARGING1 := RELAY_BAT1 AND BATTERY_CHARGING;
END_FUNCTION_BLOCK

(* POU PROGRAM_FBs/HYDRAULIC_CONTROL, LD *)
FUNCTION_BLOCK HYDRAULIC_CONTROL
VAR_INPUT
	DEADMAN: BOOL;
END_VAR
VAR_OUTPUT
END_VAR
VAR
	HYD_SPEED: INT;
	IDLE_MODE: BOOL;
	CUTOFF: INT;
	STATISTICS: STATISTICS_INT;
	RESET_AVG: BOOL;
	T1: TON;
	TRIG_1: R_TRIG;
	T2: TON;
	RUNNING_AVG: INT:=0;
	SET_IDLE: BOOL;
	HIGH_RPM: BOOL;
	WAIT: BOOL;
	UPPER_LIMIT: INT;
	MCU_RX_6: CHARA_MCU_RX;
	MCU_TX_6: CHARA_MCU_TX;
END_VAR
VAR CONSTANT
	IDLE_SPEED: INT :=0;
	ECO_CUTOFF: INT := 70;
	POWER_CUTOFF: INT := 90;
	BUFFER: INT := 10;
	HYD_RAMP: INT:= 100;
	MCU_RAMP: BYTE := 5;
	PHASE_LIMIT: BYTE := 60;
END_VAR
